LIN {X 0,Y 406.428,Z 396.116,A -85,B 0,C 180,E1 17978.8,E2 17978.8} C_VEL
LIN {X 0,Y 408.276,Z 399.712,A -85,B 0,C 180,E1 17977.389,E2 17977.389} C_VEL
LIN {X 0,Y 411.856,Z 402.645,A -85,B 0,C 180,E1 17975.473,E2 17975.473} C_VEL
LIN {X 0,Y 414.278,Z 406.426,A -85,B 0,C 180,E1 17974.252,E2 17974.252} C_VEL
LIN {X 0,Y 416.644,Z 408.719,A -85,B 0,C 180,E1 17973.259,E2 17973.259} C_VEL
LIN {X 0,Y 420.794,Z 414.411,A -85,B 0,C 180,E1 17971.588,E2 17971.588} C_VEL
LIN {X 0,Y 424.606,Z 419.568,A -85,B 0,C 180,E1 17970.247,E2 17970.247} C_VEL
LIN {X 0,Y 430.468,Z 427.804,A -85,B 0,C 180,E1 17968.376,E2 17968.376} C_VEL
LIN {X 0,Y 437.911,Z 439.101,A -85,B 0,C 180,E1 17966.262,E2 17966.262} C_VEL
LIN {X 0,Y 445.629,Z 451.395,A -85,B 0,C 180,E1 17964.313,E2 17964.313} C_VEL
LIN {X 0,Y 451.863,Z 462.203,A -85,B 0,C 180,E1 17962.861,E2 17962.861} C_VEL
LIN {X 0,Y 443.06,Z 655.512,A -85,B 0,C 180,E1 17959.181,E2 17959.181} C_VEL
LIN {X 0,Y 439.484,Z 737.589,A -85,B 0,C 180,E1 17957.617,E2 17957.617} C_VEL
LIN {X 0,Y 437.318,Z 760.996,A -85,B 0,C 180,E1 17956.985,E2 17956.985} C_VEL
LIN {X 0,Y 434.644,Z 783.7,A -85,B 0,C 180,E1 17956.155,E2 17956.155} C_VEL
LIN {X 0,Y 431.569,Z 804.772,A -85,B 0,C 180,E1 17955.152,E2 17955.152} C_VEL
LIN {X 0,Y 427.742,Z 827.839,A -85,B 0,C 180,E1 17953.785,E2 17953.785} C_VEL
LIN {X 0,Y 424.132,Z 847.133,A -85,B 0,C 180,E1 17952.397,E2 17952.397} C_VEL
LIN {X 0,Y 419.735,Z 868.682,A -85,B 0,C 180,E1 17950.546,E2 17950.546} C_VEL
LIN {X 0,Y 415.658,Z 887.581,A -85,B 0,C 180,E1 17948.629,E2 17948.629} C_VEL
LIN {X 0,Y 411.63,Z 905.465,A -85,B 0,C 180,E1 17946.487,E2 17946.487} C_VEL
LIN {X 0,Y 407.694,Z 922.843,A -85,B 0,C 180,E1 17944.086,E2 17944.086} C_VEL
LIN {X 0,Y 404.06,Z 938.881,A -85,B 0,C 180,E1 17941.479,E2 17941.479} C_VEL
LIN {X 0,Y 400.612,Z 954.751,A -85,B 0,C 180,E1 17938.474,E2 17938.474} C_VEL
LIN {X 0,Y 398,Z 967.71,A -85,B 0,C 180,E1 17935.605,E2 17935.605} C_VEL
LIN {X 0,Y 395.868,Z 979.3,A -85,B 0,C 180,E1 17932.58,E2 17932.58} C_VEL
LIN {X 0,Y 394.308,Z 989.212,A -85,B 0,C 180,E1 17929.559,E2 17929.559} C_VEL
LIN {X 0,Y 393.186,Z 997.751,A -85,B 0,C 180,E1 17926.4,E2 17926.4} C_VEL
LIN {X 0,Y 392.495,Z 1004.747,A -85,B 0,C 180,E1 17923.258,E2 17923.258} C_VEL
LIN {X 0,Y 392.089,Z 1010.305,A -85,B 0,C 180,E1 17919.99,E2 17919.99} C_VEL
LIN {X 0,Y 391.942,Z 1013.857,A -85,B 0,C 180,E1 17917.185,E2 17917.185} C_VEL
LIN {X 0,Y 391.914,Z 1016.519,A -85,B 0,C 180,E1 17913.954,E2 17913.954} C_VEL
LIN {X 0,Y 391.905,Z 1017.533,A -85,B 0,C 180,E1 17911.174,E2 17911.174} C_VEL
LIN {X 0,Y 391.911,Z 1017.466,A -85,B 0,C 180,E1 17908.396,E2 17908.396} C_VEL
LIN {X 0,Y 391.918,Z 1015.846,A -85,B 0,C 180,E1 17905.029,E2 17905.029} C_VEL
LIN {X 0,Y 391.977,Z 1013.229,A -85,B 0,C 180,E1 17902.235,E2 17902.235} C_VEL
LIN {X 0,Y 392.181,Z 1009.071,A -85,B 0,C 180,E1 17899.13,E2 17899.13} C_VEL
LIN {X 0,Y 392.616,Z 1003.242,A -85,B 0,C 180,E1 17895.993,E2 17895.993} C_VEL
LIN {X 0,Y 393.401,Z 996.051,A -85,B 0,C 180,E1 17892.858,E2 17892.858} C_VEL
LIN {X 0,Y 394.64,Z 987.03,A -85,B 0,C 180,E1 17889.695,E2 17889.695} C_VEL
LIN {X 0,Y 396.359,Z 976.876,A -85,B 0,C 180,E1 17886.667,E2 17886.667} C_VEL
LIN {X 0,Y 398.648,Z 964.781,A -85,B 0,C 180,E1 17883.651,E2 17883.651} C_VEL
LIN {X 0,Y 401.452,Z 951.514,A -85,B 0,C 180,E1 17880.787,E2 17880.787} C_VEL
LIN {X 0,Y 404.687,Z 936.825,A -85,B 0,C 180,E1 17878.087,E2 17878.087} C_VEL
LIN {X 0,Y 408.687,Z 919.41,A -85,B 0,C 180,E1 17875.339,E2 17875.339} C_VEL
LIN {X 0,Y 412.435,Z 903.112,A -85,B 0,C 180,E1 17873.13,E2 17873.13} C_VEL
LIN {X 0,Y 416.65,Z 884.299,A -85,B 0,C 180,E1 17870.951,E2 17870.951} C_VEL
LIN {X 0,Y 420.873,Z 864.938,A -85,B 0,C 180,E1 17869.036,E2 17869.036} C_VEL
LIN {X 0,Y 424.917,Z 844.471,A -85,B 0,C 180,E1 17867.345,E2 17867.345} C_VEL
LIN {X 0,Y 428.827,Z 823.074,A -85,B 0,C 180,E1 17865.862,E2 17865.862} C_VEL
LIN {X 0,Y 432.119,Z 802.52,A -85,B 0,C 180,E1 17864.7,E2 17864.7} C_VEL
LIN {X 0,Y 435.408,Z 778.669,A -85,B 0,C 180,E1 17863.628,E2 17863.628} C_VEL
LIN {X 0,Y 437.702,Z 758.039,A -85,B 0,C 180,E1 17862.917,E2 17862.917} C_VEL
LIN {X 0,Y 439.633,Z 733.719,A -85,B 0,C 180,E1 17862.311,E2 17862.311} C_VEL
LIN {X 0,Y 448.195,Z 525.035,A -85,B 0,C 180,E1 17858.416,E2 17858.416} C_VEL
LIN {X 0,Y 450.801,Z 461.932,A -85,B 0,C 180,E1 17857.207,E2 17857.207} C_VEL
LIN {X 0,Y 440.409,Z 445.676,A -85,B 0,C 180,E1 17855.016,E2 17855.016} C_VEL
LIN {X 0,Y 429.506,Z 429.721,A -85,B 0,C 180,E1 17852.53,E2 17852.53} C_VEL
LIN {X 0,Y 418.728,Z 414.832,A -85,B 0,C 180,E1 17849.819,E2 17849.819} C_VEL
LIN {X 0,Y 410.778,Z 404.455,A -85,B 0,C 180,E1 17847.625,E2 17847.625} C_VEL
LIN {X 0,Y 406.148,Z 398.624,A -85,B 0,C 180,E1 17846.263,E2 17846.263} C_VEL
LIN {X 0,Y 402.102,Z 393.64,A -85,B 0,C 180,E1 17845.006,E2 17845.006} C_VEL
LIN {X 0,Y 398.857,Z 389.644,A -85,B 0,C 180,E1 17843.96,E2 17843.96} C_VEL
LIN {X 0,Y 397.676,Z 388.128,A -85,B 0,C 180,E1 17843.563,E2 17843.563} C_VEL
LIN {X 0,Y 394.873,Z 385.623,A -85,B 0,C 180,E1 17842.636,E2 17842.636} C_VEL
LIN {X 0,Y 393.655,Z 382.808,A -85,B 0,C 180,E1 17842.034,E2 17842.034} C_VEL
LIN {X 0,Y 393.526,Z 382.083,A -85,B 0,C 180,E1 17841.461,E2 17841.461} C_VEL
LIN {X 0,Y 393.528,Z 382.017,A -85,B 0,C 180,E1 17837.446,E2 17837.446} C_VEL
LIN {X 0,Y 393.545,Z 382.024,A -85,B 0,C 180,E1 17833.517,E2 17833.517} C_VEL
LIN {X 0,Y 393.537,Z 382.019,A -85,B 0,C 180,E1 17829.505,E2 17829.505} C_VEL
LIN {X 0,Y 393.517,Z 382.017,A -85,B 0,C 180,E1 17825.686,E2 17825.686} C_VEL
LIN {X 0,Y 393.511,Z 382.017,A -85,B 0,C 180,E1 17821.747,E2 17821.747} C_VEL
LIN {X 0,Y 393.504,Z 382.024,A -85,B 0,C 180,E1 17817.961,E2 17817.961} C_VEL
LIN {X 0,Y 393.507,Z 382.031,A -85,B 0,C 180,E1 17814.02,E2 17814.02} C_VEL
LIN {X 0,Y 393.514,Z 382.03,A -85,B 0,C 180,E1 17810.05,E2 17810.05} C_VEL
LIN {X 0,Y 393.528,Z 382.024,A -85,B 0,C 180,E1 17806.182,E2 17806.182} C_VEL
LIN {X 0,Y 393.545,Z 382.014,A -85,B 0,C 180,E1 17802.294,E2 17802.294} C_VEL
LIN {X 0,Y 393.567,Z 382.01,A -85,B 0,C 180,E1 17798.384,E2 17798.384} C_VEL
LIN {X 0,Y 393.56,Z 382.013,A -85,B 0,C 180,E1 17794.393,E2 17794.393} C_VEL
LIN {X 0,Y 393.558,Z 382.018,A -85,B 0,C 180,E1 17790.47,E2 17790.47} C_VEL
LIN {X 0,Y 393.546,Z 382.028,A -85,B 0,C 180,E1 17786.542,E2 17786.542} C_VEL
LIN {X 0,Y 393.537,Z 382.019,A -85,B 0,C 180,E1 17782.61,E2 17782.61} C_VEL
LIN {X 0,Y 393.532,Z 382.015,A -85,B 0,C 180,E1 17778.759,E2 17778.759} C_VEL
LIN {X 0,Y 393.533,Z 382.024,A -85,B 0,C 180,E1 17774.723,E2 17774.723} C_VEL
LIN {X 0,Y 393.534,Z 382.018,A -85,B 0,C 180,E1 17770.758,E2 17770.758} C_VEL
LIN {X 0,Y 393.613,Z 382.321,A -85,B 0,C 180,E1 17769.416,E2 17769.416} C_VEL
LIN {X 0,Y 393.952,Z 383.729,A -85,B 0,C 180,E1 17769.046,E2 17769.046} C_VEL
LIN {X 0,Y 395.637,Z 386.503,A -85,B 0,C 180,E1 17768.423,E2 17768.423} C_VEL
LIN {X 0,Y 398.831,Z 388.927,A -85,B 0,C 180,E1 17767.401,E2 17767.401} C_VEL
LIN {X 0,Y 401.009,Z 392.541,A -85,B 0,C 180,E1 17766.655,E2 17766.655} C_VEL
LIN {X 0,Y 404.151,Z 395.276,A -85,B 0,C 180,E1 17765.715,E2 17765.715} C_VEL
LIN {X 0,Y 406.926,Z 399.204,A -85,B 0,C 180,E1 17764.847,E2 17764.847} C_VEL
LIN {X 0,Y 409.166,Z 401.398,A -85,B 0,C 180,E1 17764.205,E2 17764.205} C_VEL
LIN {X 0,Y 412.49,Z 405.713,A -85,B 0,C 180,E1 17763.251,E2 17763.251} C_VEL
LIN {X 0,Y 414.192,Z 407.663,A -85,B 0,C 180,E1 17762.788,E2 17762.788} C_VEL
LIN {X 0,Y 419.544,Z 414.327,A -85,B 0,C 180,E1 17761.373,E2 17761.373} C_VEL
LIN {X 0,Y 423.817,Z 419.73,A -85,B 0,C 180,E1 17760.292,E2 17760.292} C_VEL
LIN {X 0,Y 432.407,Z 430.894,A -85,B 0,C 180,E1 17758.237,E2 17758.237} C_VEL
LIN {X 0,Y 443.538,Z 446.105,A -85,B 0,C 180,E1 17755.797,E2 17755.797} C_VEL
LIN {X 0,Y 450.635,Z 456.669,A -85,B 0,C 180,E1 17754.337,E2 17754.337} C_VEL
LIN {X 0,Y 441.914,Z 664.576,A -85,B 0,C 180,E1 17750.46,E2 17750.46} C_VEL
LIN {X 0,Y 441.065,Z 686.182,A -85,B 0,C 180,E1 17750.061,E2 17750.061} C_VEL
LIN {X 0,Y 440.083,Z 693.883,A -85,B 0,C 180,E1 17750.016,E2 17750.016} C_VEL
LIN {X 0,Y 434.779,Z 714.411,A -85,B 0,C 180,E1 17750.219,E2 17750.219} C_VEL
LIN {X 0,Y 433.809,Z 720.955,A -85,B 0,C 180,E1 17750.126,E2 17750.126} C_VEL
LIN {X 0,Y 431.867,Z 741.999,A -85,B 0,C 180,E1 17749.509,E2 17749.509} C_VEL
LIN {X 0,Y 429.108,Z 764.775,A -85,B 0,C 180,E1 17748.611,E2 17748.611} C_VEL
LIN {X 0,Y 426.34,Z 783.59,A -85,B 0,C 180,E1 17747.675,E2 17747.675} C_VEL
LIN {X 0,Y 422.604,Z 805.364,A -85,B 0,C 180,E1 17746.348,E2 17746.348} C_VEL
LIN {X 0,Y 419.031,Z 823.676,A -85,B 0,C 180,E1 17745,E2 17745} C_VEL
LIN {X 0,Y 414.557,Z 844.411,A -85,B 0,C 180,E1 17743.183,E2 17743.183} C_VEL
LIN {X 0,Y 410.383,Z 862.505,A -85,B 0,C 180,E1 17741.306,E2 17741.306} C_VEL
LIN {X 0,Y 406.042,Z 880.264,A -85,B 0,C 180,E1 17739.134,E2 17739.134} C_VEL
LIN {X 0,Y 402.007,Z 896.346,A -85,B 0,C 180,E1 17736.852,E2 17736.852} C_VEL
LIN {X 0,Y 398.055,Z 911.792,A -85,B 0,C 180,E1 17734.275,E2 17734.275} C_VEL
LIN {X 0,Y 394.61,Z 925.735,A -85,B 0,C 180,E1 17731.593,E2 17731.593} C_VEL
LIN {X 0,Y 391.538,Z 938.518,A -85,B 0,C 180,E1 17728.679,E2 17728.679} C_VEL
LIN {X 0,Y 388.972,Z 950.224,A -85,B 0,C 180,E1 17725.573,E2 17725.573} C_VEL
LIN {X 0,Y 387.022,Z 960.112,A -85,B 0,C 180,E1 17722.425,E2 17722.425} C_VEL
LIN {X 0,Y 385.538,Z 969.205,A -85,B 0,C 180,E1 17718.931,E2 17718.931} C_VEL
LIN {X 0,Y 384.68,Z 975.978,A -85,B 0,C 180,E1 17715.7,E2 17715.7} C_VEL
LIN {X 0,Y 384.188,Z 981.504,A -85,B 0,C 180,E1 17712.268,E2 17712.268} C_VEL
LIN {X 0,Y 383.982,Z 985.352,A -85,B 0,C 180,E1 17708.936,E2 17708.936} C_VEL
LIN {X 0,Y 383.929,Z 987.716,A -85,B 0,C 180,E1 17705.535,E2 17705.535} C_VEL
LIN {X 0,Y 383.908,Z 988.577,A -85,B 0,C 180,E1 17702.315,E2 17702.315} C_VEL
LIN {X 0,Y 383.929,Z 987.981,A -85,B 0,C 180,E1 17698.955,E2 17698.955} C_VEL
LIN {X 0,Y 383.955,Z 985.95,A -85,B 0,C 180,E1 17695.588,E2 17695.588} C_VEL
LIN {X 0,Y 384.133,Z 982.409,A -85,B 0,C 180,E1 17692.285,E2 17692.285} C_VEL
LIN {X 0,Y 384.541,Z 977.393,A -85,B 0,C 180,E1 17688.942,E2 17688.942} C_VEL
LIN {X 0,Y 385.364,Z 970.543,A -85,B 0,C 180,E1 17685.522,E2 17685.522} C_VEL
LIN {X 0,Y 386.671,Z 962.482,A -85,B 0,C 180,E1 17682.247,E2 17682.247} C_VEL
LIN {X 0,Y 388.536,Z 952.579,A -85,B 0,C 180,E1 17678.994,E2 17678.994} C_VEL
LIN {X 0,Y 391.128,Z 940.768,A -85,B 0,C 180,E1 17675.723,E2 17675.723} C_VEL
LIN {X 0,Y 394.033,Z 928.538,A -85,B 0,C 180,E1 17672.865,E2 17672.865} C_VEL
LIN {X 0,Y 397.816,Z 913.455,A -85,B 0,C 180,E1 17669.87,E2 17669.87} C_VEL
LIN {X 0,Y 401.794,Z 898.064,A -85,B 0,C 180,E1 17667.251,E2 17667.251} C_VEL
LIN {X 0,Y 405.906,Z 881.802,A -85,B 0,C 180,E1 17664.912,E2 17664.912} C_VEL
LIN {X 0,Y 410.309,Z 864.198,A -85,B 0,C 180,E1 17662.721,E2 17662.721} C_VEL
LIN {X 0,Y 414.446,Z 846.464,A -85,B 0,C 180,E1 17660.853,E2 17660.853} C_VEL
LIN {X 0,Y 418.988,Z 825.858,A -85,B 0,C 180,E1 17659.011,E2 17659.011} C_VEL
LIN {X 0,Y 422.741,Z 806.937,A -85,B 0,C 180,E1 17657.598,E2 17657.598} C_VEL
LIN {X 0,Y 426.635,Z 784.75,A -85,B 0,C 180,E1 17656.229,E2 17656.229} C_VEL
LIN {X 0,Y 429.41,Z 766.27,A -85,B 0,C 180,E1 17655.298,E2 17655.298} C_VEL
LIN {X 0,Y 432.256,Z 743.229,A -85,B 0,C 180,E1 17654.377,E2 17654.377} C_VEL
LIN {X 0,Y 434.174,Z 722.916,A -85,B 0,C 180,E1 17653.771,E2 17653.771} C_VEL
LIN {X 0,Y 435.95,Z 691.902,A -85,B 0,C 180,E1 17653.119,E2 17653.119} C_VEL
LIN {X 0,Y 445.434,Z 492.104,A -85,B 0,C 180,E1 17649.297,E2 17649.297} C_VEL
LIN {X 0,Y 446.947,Z 460.775,A -85,B 0,C 180,E1 17648.669,E2 17648.669} C_VEL
LIN {X 0,Y 438.774,Z 448.403,A -85,B 0,C 180,E1 17646.674,E2 17646.674} C_VEL
LIN {X 0,Y 430.575,Z 436.674,A -85,B 0,C 180,E1 17644.429,E2 17644.429} C_VEL
LIN {X 0,Y 425.629,Z 430.22,A -85,B 0,C 180,E1 17642.916,E2 17642.916} C_VEL
LIN {X 0,Y 422.462,Z 426.015,A -85,B 0,C 180,E1 17641.865,E2 17641.865} C_VEL
LIN {X 0,Y 418.675,Z 421.042,A -85,B 0,C 180,E1 17640.479,E2 17640.479} C_VEL
LIN {X 0,Y 415.228,Z 416.743,A -85,B 0,C 180,E1 17639.104,E2 17639.104} C_VEL
LIN {X 0,Y 414.077,Z 415.376,A -85,B 0,C 180,E1 17638.608,E2 17638.608} C_VEL
LIN {X 0,Y 410.92,Z 411.698,A -85,B 0,C 180,E1 17637.107,E2 17637.107} C_VEL
LIN {X 0,Y 409.736,Z 409.74,A -85,B 0,C 180,E1 17636.465,E2 17636.465} C_VEL
LIN {X 0,Y 406.459,Z 406.882,A -85,B 0,C 180,E1 17634.566,E2 17634.566} C_VEL
LIN {X 0,Y 404.667,Z 403.582,A -85,B 0,C 180,E1 17633.189,E2 17633.189} C_VEL
LIN {X 0,Y 400.609,Z 400.405,A -85,B 0,C 180,E1 17628.483,E2 17628.483} C_VEL
LIN {X 0,Y 400.207,Z 399.651,A -85,B 0,C 180,E1 17625.976,E2 17625.976} C_VEL
LIN {X 0,Y 400.964,Z 400.936,A -85,B 0,C 180,E1 17623.187,E2 17623.187} C_VEL
LIN {X 0,Y 405.042,Z 404.041,A -85,B 0,C 180,E1 17618.985,E2 17618.985} C_VEL
LIN {X 0,Y 406.914,Z 407.563,A -85,B 0,C 180,E1 17617.53,E2 17617.53} C_VEL
LIN {X 0,Y 410.102,Z 410.218,A -85,B 0,C 180,E1 17615.783,E2 17615.783} C_VEL
LIN {X 0,Y 412.806,Z 414.296,A -85,B 0,C 180,E1 17614.384,E2 17614.384} C_VEL
LIN {X 0,Y 414.826,Z 416.366,A -85,B 0,C 180,E1 17613.519,E2 17613.519} C_VEL
LIN {X 0,Y 418.809,Z 421.973,A -85,B 0,C 180,E1 17611.868,E2 17611.868} C_VEL
LIN {X 0,Y 422.265,Z 426.738,A -85,B 0,C 180,E1 17610.616,E2 17610.616} C_VEL
LIN {X 0,Y 427.794,Z 434.728,A -85,B 0,C 180,E1 17608.784,E2 17608.784} C_VEL
LIN {X 0,Y 435.211,Z 446.196,A -85,B 0,C 180,E1 17606.618,E2 17606.618} C_VEL
LIN {X 0,Y 443.39,Z 459.583,A -85,B 0,C 180,E1 17604.499,E2 17604.499} C_VEL
LIN {X 0,Y 447.005,Z 466.235,A -85,B 0,C 180,E1 17603.619,E2 17603.619} C_VEL
LIN {X 0,Y 437.783,Z 657.986,A -85,B 0,C 180,E1 17599.933,E2 17599.933} C_VEL
LIN {X 0,Y 434.097,Z 737.688,A -85,B 0,C 180,E1 17598.396,E2 17598.396} C_VEL
LIN {X 0,Y 431.819,Z 761.162,A -85,B 0,C 180,E1 17597.754,E2 17597.754} C_VEL
LIN {X 0,Y 428.968,Z 784.037,A -85,B 0,C 180,E1 17596.907,E2 17596.907} C_VEL
LIN {X 0,Y 425.651,Z 805.681,A -85,B 0,C 180,E1 17595.862,E2 17595.862} C_VEL
LIN {X 0,Y 421.685,Z 828.309,A -85,B 0,C 180,E1 17594.499,E2 17594.499} C_VEL
LIN {X 0,Y 417.893,Z 847.639,A -85,B 0,C 180,E1 17593.089,E2 17593.089} C_VEL
LIN {X 0,Y 413.338,Z 868.814,A -85,B 0,C 180,E1 17591.24,E2 17591.24} C_VEL
LIN {X 0,Y 409.022,Z 887.843,A -85,B 0,C 180,E1 17589.285,E2 17589.285} C_VEL
LIN {X 0,Y 404.67,Z 906.087,A -85,B 0,C 180,E1 17587.055,E2 17587.055} C_VEL
LIN {X 0,Y 400.525,Z 923.381,A -85,B 0,C 180,E1 17584.609,E2 17584.609} C_VEL
LIN {X 0,Y 396.9,Z 938.465,A -85,B 0,C 180,E1 17582.114,E2 17582.114} C_VEL
LIN {X 0,Y 393.234,Z 954.35,A -85,B 0,C 180,E1 17579.059,E2 17579.059} C_VEL
LIN {X 0,Y 390.582,Z 966.668,A -85,B 0,C 180,E1 17576.291,E2 17576.291} C_VEL
LIN {X 0,Y 388.169,Z 978.931,A -85,B 0,C 180,E1 17573.053,E2 17573.053} C_VEL
LIN {X 0,Y 386.49,Z 988.853,A -85,B 0,C 180,E1 17569.971,E2 17569.971} C_VEL
LIN {X 0,Y 385.283,Z 997.406,A -85,B 0,C 180,E1 17566.746,E2 17566.746} C_VEL
LIN {X 0,Y 384.564,Z 1004.101,A -85,B 0,C 180,E1 17563.69,E2 17563.69} C_VEL
LIN {X 0,Y 384.113,Z 1009.865,A -85,B 0,C 180,E1 17560.284,E2 17560.284} C_VEL
LIN {X 0,Y 383.956,Z 1013.377,A -85,B 0,C 180,E1 17557.486,E2 17557.486} C_VEL
LIN {X 0,Y 383.918,Z 1016.142,A -85,B 0,C 180,E1 17554.186,E2 17554.186} C_VEL
LIN {X 0,Y 383.911,Z 1017.231,A -85,B 0,C 180,E1 17551.198,E2 17551.198} C_VEL
LIN {X 0,Y 383.916,Z 1017.167,A -85,B 0,C 180,E1 17548.363,E2 17548.363} C_VEL
LIN {X 0,Y 383.923,Z 1015.548,A -85,B 0,C 180,E1 17544.925,E2 17544.925} C_VEL
LIN {X 0,Y 384.008,Z 1012.766,A -85,B 0,C 180,E1 17541.922,E2 17541.922} C_VEL
LIN {X 0,Y 384.239,Z 1007.992,A -85,B 0,C 180,E1 17538.447,E2 17538.447} C_VEL
LIN {X 0,Y 384.73,Z 1002.337,A -85,B 0,C 180,E1 17535.404,E2 17535.404} C_VEL
LIN {X 0,Y 385.685,Z 994.537,A -85,B 0,C 180,E1 17532.037,E2 17532.037} C_VEL
LIN {X 0,Y 387.024,Z 985.772,A -85,B 0,C 180,E1 17528.961,E2 17528.961} C_VEL
LIN {X 0,Y 389.148,Z 974.254,A -85,B 0,C 180,E1 17525.571,E2 17525.571} C_VEL
LIN {X 0,Y 391.585,Z 962.5,A -85,B 0,C 180,E1 17522.645,E2 17522.645} C_VEL
LIN {X 0,Y 394.843,Z 948.018,A -85,B 0,C 180,E1 17519.578,E2 17519.578} C_VEL
LIN {X 0,Y 398.536,Z 932.669,A -85,B 0,C 180,E1 17516.787,E2 17516.787} C_VEL
LIN {X 0,Y 402.43,Z 916.445,A -85,B 0,C 180,E1 17514.284,E2 17514.284} C_VEL
LIN {X 0,Y 406.754,Z 898.616,A -85,B 0,C 180,E1 17511.91,E2 17511.91} C_VEL
LIN {X 0,Y 410.829,Z 881.207,A -85,B 0,C 180,E1 17509.937,E2 17509.937} C_VEL
LIN {X 0,Y 415.463,Z 860.345,A -85,B 0,C 180,E1 17507.922,E2 17507.922} C_VEL
LIN {X 0,Y 419.428,Z 841.214,A -85,B 0,C 180,E1 17506.368,E2 17506.368} C_VEL
LIN {X 0,Y 423.486,Z 819.472,A -85,B 0,C 180,E1 17504.905,E2 17504.905} C_VEL
LIN {X 0,Y 427.068,Z 797.92,A -85,B 0,C 180,E1 17503.718,E2 17503.718} C_VEL
LIN {X 0,Y 430.038,Z 776.108,A -85,B 0,C 180,E1 17502.776,E2 17502.776} C_VEL
LIN {X 0,Y 432.538,Z 754.231,A -85,B 0,C 180,E1 17502.042,E2 17502.042} C_VEL
LIN {X 0,Y 434.294,Z 730.724,A -85,B 0,C 180,E1 17501.484,E2 17501.484} C_VEL
LIN {X 0,Y 443.269,Z 521.692,A -85,B 0,C 180,E1 17497.553,E2 17497.553} C_VEL
LIN {X 0,Y 445.703,Z 465.789,A -85,B 0,C 180,E1 17496.475,E2 17496.475} C_VEL
LIN {X 0,Y 435.041,Z 449.15,A -85,B 0,C 180,E1 17494.149,E2 17494.149} C_VEL
LIN {X 0,Y 425.183,Z 434.788,A -85,B 0,C 180,E1 17491.826,E2 17491.826} C_VEL
LIN {X 0,Y 415.533,Z 421.274,A -85,B 0,C 180,E1 17489.318,E2 17489.318} C_VEL
LIN {X 0,Y 407.875,Z 411.22,A -85,B 0,C 180,E1 17487.165,E2 17487.165} C_VEL
LIN {X 0,Y 403.321,Z 405.407,A -85,B 0,C 180,E1 17485.789,E2 17485.789} C_VEL
LIN {X 0,Y 399.612,Z 400.791,A -85,B 0,C 180,E1 17484.619,E2 17484.619} C_VEL
LIN {X 0,Y 395.945,Z 396.037,A -85,B 0,C 180,E1 17483.396,E2 17483.396} C_VEL
LIN {X 0,Y 392.41,Z 392.601,A -85,B 0,C 180,E1 17482.193,E2 17482.193} C_VEL
LIN {X 0,Y 390.723,Z 389.598,A -85,B 0,C 180,E1 17481.543,E2 17481.543} C_VEL
LIN {X 0,Y 387.439,Z 387.253,A -85,B 0,C 180,E1 17480.388,E2 17480.388} C_VEL
LIN {X 0,Y 385.72,Z 383.756,A -85,B 0,C 180,E1 17479.535,E2 17479.535} C_VEL
LIN {X 0,Y 385.558,Z 383.051,A -85,B 0,C 180,E1 17478.914,E2 17478.914} C_VEL
LIN {X 0,Y 385.565,Z 383.008,A -85,B 0,C 180,E1 17475.029,E2 17475.029} C_VEL
LIN {X 0,Y 385.588,Z 383.006,A -85,B 0,C 180,E1 17471.214,E2 17471.214} C_VEL
LIN {X 0,Y 385.602,Z 383.015,A -85,B 0,C 180,E1 17467.149,E2 17467.149} C_VEL
LIN {X 0,Y 385.602,Z 383.008,A -85,B 0,C 180,E1 17463.121,E2 17463.121} C_VEL
LIN {X 0,Y 385.614,Z 383.001,A -85,B 0,C 180,E1 17459.108,E2 17459.108} C_VEL
LIN {X 0,Y 385.606,Z 383.003,A -85,B 0,C 180,E1 17455.091,E2 17455.091} C_VEL
LIN {X 0,Y 385.595,Z 383.006,A -85,B 0,C 180,E1 17451.199,E2 17451.199} C_VEL
LIN {X 0,Y 385.586,Z 383.015,A -85,B 0,C 180,E1 17447.266,E2 17447.266} C_VEL
LIN {X 0,Y 385.578,Z 383.02,A -85,B 0,C 180,E1 17443.426,E2 17443.426} C_VEL
LIN {X 0,Y 385.58,Z 383.014,A -85,B 0,C 180,E1 17439.391,E2 17439.391} C_VEL
LIN {X 0,Y 385.579,Z 383.006,A -85,B 0,C 180,E1 17435.323,E2 17435.323} C_VEL
LIN {X 0,Y 385.583,Z 383.003,A -85,B 0,C 180,E1 17431.332,E2 17431.332} C_VEL
LIN {X 0,Y 385.589,Z 383.01,A -85,B 0,C 180,E1 17427.359,E2 17427.359} C_VEL
LIN {X 0,Y 385.597,Z 383.018,A -85,B 0,C 180,E1 17423.387,E2 17423.387} C_VEL
LIN {X 0,Y 385.605,Z 383.004,A -85,B 0,C 180,E1 17419.395,E2 17419.395} C_VEL
LIN {X 0,Y 385.61,Z 383.003,A -85,B 0,C 180,E1 17415.357,E2 17415.357} C_VEL
LIN {X 0,Y 385.661,Z 383.299,A -85,B 0,C 180,E1 17411.973,E2 17411.973} C_VEL
LIN {X 0,Y 386.02,Z 384.671,A -85,B 0,C 180,E1 17411.527,E2 17411.527} C_VEL
LIN {X 0,Y 387.738,Z 387.532,A -85,B 0,C 180,E1 17410.812,E2 17410.812} C_VEL
LIN {X 0,Y 391.046,Z 389.934,A -85,B 0,C 180,E1 17409.65,E2 17409.65} C_VEL
LIN {X 0,Y 393.067,Z 393.427,A -85,B 0,C 180,E1 17408.886,E2 17408.886} C_VEL
LIN {X 0,Y 396.358,Z 396.252,A -85,B 0,C 180,E1 17407.799,E2 17407.799} C_VEL
LIN {X 0,Y 399.057,Z 400.215,A -85,B 0,C 180,E1 17406.879,E2 17406.879} C_VEL
LIN {X 0,Y 401.715,Z 402.679,A -85,B 0,C 180,E1 17406.069,E2 17406.069} C_VEL
LIN {X 0,Y 404.956,Z 406.856,A -85,B 0,C 180,E1 17405.065,E2 17405.065} C_VEL
LIN {X 0,Y 406.693,Z 408.75,A -85,B 0,C 180,E1 17404.552,E2 17404.552} C_VEL
LIN {X 0,Y 410.478,Z 413.367,A -85,B 0,C 180,E1 17403.459,E2 17403.459} C_VEL
LIN {X 0,Y 420.192,Z 425.608,A -85,B 0,C 180,E1 17400.866,E2 17400.866} C_VEL
LIN {X 0,Y 431.442,Z 440.478,A -85,B 0,C 180,E1 17398.138,E2 17398.138} C_VEL
LIN {X 0,Y 443.192,Z 457.042,A -85,B 0,C 180,E1 17395.559,E2 17395.559} C_VEL
LIN {X 0,Y 445.503,Z 460.776,A -85,B 0,C 180,E1 17395.069,E2 17395.069} C_VEL
LIN {X 0,Y 436.352,Z 669.306,A -85,B 0,C 180,E1 17391.15,E2 17391.15} C_VEL
LIN {X 0,Y 434.124,Z 717.19,A -85,B 0,C 180,E1 17390.223,E2 17390.223} C_VEL
LIN {X 0,Y 433.809,Z 720.955,A -85,B 0,C 180,E1 17390.126,E2 17390.126} C_VEL
LIN {X 0,Y 432.442,Z 728.564,A -85,B 0,C 180,E1 17390.036,E2 17390.036} C_VEL
LIN {X 0,Y 426.299,Z 747.731,A -85,B 0,C 180,E1 17390.024,E2 17390.024} C_VEL
LIN {X 0,Y 424.81,Z 755.185,A -85,B 0,C 180,E1 17389.809,E2 17389.809} C_VEL
LIN {X 0,Y 421.501,Z 778.336,A -85,B 0,C 180,E1 17388.744,E2 17388.744} C_VEL
LIN {X 0,Y 417.955,Z 799.173,A -85,B 0,C 180,E1 17387.538,E2 17387.538} C_VEL
LIN {X 0,Y 413.828,Z 820.109,A -85,B 0,C 180,E1 17386.055,E2 17386.055} C_VEL
LIN {X 0,Y 409.772,Z 838.808,A -85,B 0,C 180,E1 17384.479,E2 17384.479} C_VEL
LIN {X 0,Y 405.135,Z 858.13,A -85,B 0,C 180,E1 17382.539,E2 17382.539} C_VEL
LIN {X 0,Y 400.618,Z 876.151,A -85,B 0,C 180,E1 17380.42,E2 17380.42} C_VEL
LIN {X 0,Y 396.248,Z 892.644,A -85,B 0,C 180,E1 17378.119,E2 17378.119} C_VEL
LIN {X 0,Y 392.03,Z 908.525,A -85,B 0,C 180,E1 17375.557,E2 17375.557} C_VEL
LIN {X 0,Y 388.165,Z 922.99,A -85,B 0,C 180,E1 17372.801,E2 17372.801} C_VEL
LIN {X 0,Y 384.455,Z 937.496,A -85,B 0,C 180,E1 17369.548,E2 17369.548} C_VEL
LIN {X 0,Y 381.649,Z 949.412,A -85,B 0,C 180,E1 17366.391,E2 17366.391} C_VEL
LIN {X 0,Y 379.497,Z 959.438,A -85,B 0,C 180,E1 17363.187,E2 17363.187} C_VEL
LIN {X 0,Y 377.901,Z 968.388,A -85,B 0,C 180,E1 17359.785,E2 17359.785} C_VEL
LIN {X 0,Y 376.887,Z 975.289,A -85,B 0,C 180,E1 17356.495,E2 17356.495} C_VEL
LIN {X 0,Y 376.282,Z 981.105,A -85,B 0,C 180,E1 17353.001,E2 17353.001} C_VEL
LIN {X 0,Y 376.034,Z 984.954,A -85,B 0,C 180,E1 17349.774,E2 17349.774} C_VEL
LIN {X 0,Y 375.921,Z 987.6,A -85,B 0,C 180,E1 17346.483,E2 17346.483} C_VEL
LIN {X 0,Y 375.915,Z 988.737,A -85,B 0,C 180,E1 17343.284,E2 17343.284} C_VEL
LIN {X 0,Y 375.909,Z 988.705,A -85,B 0,C 180,E1 17340.344,E2 17340.344} C_VEL
LIN {X 0,Y 375.941,Z 987.282,A -85,B 0,C 180,E1 17336.907,E2 17336.907} C_VEL
LIN {X 0,Y 376.039,Z 984.684,A -85,B 0,C 180,E1 17333.819,E2 17333.819} C_VEL
LIN {X 0,Y 376.355,Z 980.422,A -85,B 0,C 180,E1 17330.382,E2 17330.382} C_VEL
LIN {X 0,Y 376.989,Z 974.724,A -85,B 0,C 180,E1 17327.056,E2 17327.056} C_VEL
LIN {X 0,Y 378.188,Z 966.823,A -85,B 0,C 180,E1 17323.425,E2 17323.425} C_VEL
LIN {X 0,Y 379.817,Z 958.221,A -85,B 0,C 180,E1 17320.229,E2 17320.229} C_VEL
LIN {X 0,Y 382.266,Z 947.064,A -85,B 0,C 180,E1 17316.797,E2 17316.797} C_VEL
LIN {X 0,Y 385.16,Z 935.351,A -85,B 0,C 180,E1 17313.748,E2 17313.748} C_VEL
LIN {X 0,Y 388.679,Z 921.716,A -85,B 0,C 180,E1 17310.768,E2 17310.768} C_VEL
LIN {X 0,Y 392.807,Z 906.532,A -85,B 0,C 180,E1 17307.928,E2 17307.928} C_VEL
LIN {X 0,Y 396.875,Z 891.423,A -85,B 0,C 180,E1 17305.519,E2 17305.519} C_VEL
LIN {X 0,Y 401.802,Z 872.874,A -85,B 0,C 180,E1 17302.998,E2 17302.998} C_VEL
LIN {X 0,Y 406.27,Z 855.442,A -85,B 0,C 180,E1 17300.983,E2 17300.983} C_VEL
LIN {X 0,Y 410.824,Z 836.233,A -85,B 0,C 180,E1 17299.108,E2 17299.108} C_VEL
LIN {X 0,Y 415.255,Z 816.101,A -85,B 0,C 180,E1 17297.445,E2 17297.445} C_VEL
LIN {X 0,Y 419.263,Z 795.229,A -85,B 0,C 180,E1 17296.032,E2 17296.032} C_VEL
LIN {X 0,Y 423.062,Z 772.693,A -85,B 0,C 180,E1 17294.789,E2 17294.789} C_VEL
LIN {X 0,Y 425.887,Z 752.197,A -85,B 0,C 180,E1 17293.895,E2 17293.895} C_VEL
LIN {X 0,Y 428.471,Z 728.496,A -85,B 0,C 180,E1 17293.109,E2 17293.109} C_VEL
LIN {X 0,Y 430.076,Z 706.892,A -85,B 0,C 180,E1 17292.596,E2 17292.596} C_VEL
LIN {X 0,Y 440.369,Z 500.943,A -85,B 0,C 180,E1 17288.617,E2 17288.617} C_VEL
LIN {X 0,Y 442.238,Z 464.937,A -85,B 0,C 180,E1 17287.894,E2 17287.894} C_VEL
LIN {X 0,Y 433.689,Z 451.973,A -85,B 0,C 180,E1 17285.69,E2 17285.69} C_VEL
LIN {X 0,Y 426.589,Z 441.93,A -85,B 0,C 180,E1 17283.629,E2 17283.629} C_VEL
LIN {X 0,Y 420.568,Z 433.629,A -85,B 0,C 180,E1 17281.635,E2 17281.635} C_VEL
LIN {X 0,Y 416.392,Z 428.208,A -85,B 0,C 180,E1 17280.069,E2 17280.069} C_VEL
LIN {X 0,Y 412.927,Z 423.552,A -85,B 0,C 180,E1 17278.613,E2 17278.613} C_VEL
LIN {X 0,Y 409.243,Z 419.35,A -85,B 0,C 180,E1 17276.849,E2 17276.849} C_VEL
LIN {X 0,Y 408.086,Z 417.423,A -85,B 0,C 180,E1 17276.208,E2 17276.208} C_VEL
LIN {X 0,Y 404.779,Z 414.277,A -85,B 0,C 180,E1 17274.188,E2 17274.188} C_VEL
LIN {X 0,Y 403.152,Z 411.298,A -85,B 0,C 180,E1 17272.877,E2 17272.877} C_VEL
LIN {X 0,Y 399.371,Z 408.062,A -85,B 0,C 180,E1 17268.007,E2 17268.007} C_VEL
LIN {X 0,Y 399.136,Z 407.651,A -85,B 0,C 180,E1 17265.641,E2 17265.641} C_VEL
LIN {X 0,Y 400.343,Z 409.394,A -85,B 0,C 180,E1 17262.411,E2 17262.411} C_VEL
LIN {X 0,Y 403.575,Z 411.758,A -85,B 0,C 180,E1 17259.251,E2 17259.251} C_VEL
LIN {X 0,Y 405.54,Z 415.384,A -85,B 0,C 180,E1 17257.686,E2 17257.686} C_VEL
LIN {X 0,Y 408.419,Z 417.888,A -85,B 0,C 180,E1 17256.061,E2 17256.061} C_VEL
LIN {X 0,Y 411.201,Z 422.009,A -85,B 0,C 180,E1 17254.586,E2 17254.586} C_VEL
LIN {X 0,Y 413.018,Z 423.995,A -85,B 0,C 180,E1 17253.781,E2 17253.781} C_VEL
LIN {X 0,Y 416.761,Z 429.392,A -85,B 0,C 180,E1 17252.185,E2 17252.185} C_VEL
LIN {X 0,Y 420.139,Z 434.206,A -85,B 0,C 180,E1 17250.917,E2 17250.917} C_VEL
LIN {X 0,Y 425.268,Z 441.814,A -85,B 0,C 180,E1 17249.167,E2 17249.167} C_VEL
LIN {X 0,Y 432.638,Z 453.448,A -85,B 0,C 180,E1 17246.948,E2 17246.948} C_VEL
LIN {X 0,Y 441.399,Z 468.266,A -85,B 0,C 180,E1 17244.623,E2 17244.623} C_VEL
LIN {X 0,Y 442.267,Z 470.23,A -85,B 0,C 180,E1 17244.396,E2 17244.396} C_VEL
LIN {X 0,Y 432.512,Z 662.131,A -85,B 0,C 180,E1 17240.672,E2 17240.672} C_VEL
LIN {X 0,Y 428.854,Z 737.152,A -85,B 0,C 180,E1 17239.21,E2 17239.21} C_VEL
LIN {X 0,Y 426.51,Z 760.474,A -85,B 0,C 180,E1 17238.571,E2 17238.571} C_VEL
LIN {X 0,Y 423.635,Z 782.793,A -85,B 0,C 180,E1 17237.749,E2 17237.749} C_VEL
LIN {X 0,Y 420.237,Z 804.101,A -85,B 0,C 180,E1 17236.727,E2 17236.727} C_VEL
LIN {X 0,Y 416.245,Z 826.089,A -85,B 0,C 180,E1 17235.419,E2 17235.419} C_VEL
LIN {X 0,Y 412.088,Z 846.347,A -85,B 0,C 180,E1 17233.946,E2 17233.946} C_VEL
LIN {X 0,Y 407.317,Z 867.682,A -85,B 0,C 180,E1 17232.082,E2 17232.082} C_VEL
LIN {X 0,Y 402.928,Z 886.074,A -85,B 0,C 180,E1 17230.183,E2 17230.183} C_VEL
LIN {X 0,Y 398.333,Z 904.393,A -85,B 0,C 180,E1 17227.954,E2 17227.954} C_VEL
LIN {X 0,Y 394.03,Z 921.537,A -85,B 0,C 180,E1 17225.531,E2 17225.531} C_VEL
LIN {X 0,Y 390.008,Z 937.199,A -85,B 0,C 180,E1 17222.926,E2 17222.926} C_VEL
LIN {X 0,Y 386.455,Z 951.796,A -85,B 0,C 180,E1 17220.131,E2 17220.131} C_VEL
LIN {X 0,Y 383.356,Z 964.975,A -85,B 0,C 180,E1 17217.161,E2 17217.161} C_VEL
LIN {X 0,Y 380.7,Z 977.499,A -85,B 0,C 180,E1 17213.861,E2 17213.861} C_VEL
LIN {X 0,Y 378.919,Z 987.073,A -85,B 0,C 180,E1 17210.873,E2 17210.873} C_VEL
LIN {X 0,Y 377.435,Z 996.698,A -85,B 0,C 180,E1 17207.264,E2 17207.264} C_VEL
LIN {X 0,Y 376.665,Z 1003.14,A -85,B 0,C 180,E1 17204.296,E2 17204.296} C_VEL
LIN {X 0,Y 376.163,Z 1009.234,A -85,B 0,C 180,E1 17200.727,E2 17200.727} C_VEL
LIN {X 0,Y 375.981,Z 1012.899,A -85,B 0,C 180,E1 17197.799,E2 17197.799} C_VEL
LIN {X 0,Y 375.918,Z 1015.681,A -85,B 0,C 180,E1 17194.581,E2 17194.581} C_VEL
LIN {X 0,Y 375.921,Z 1016.905,A -85,B 0,C 180,E1 17191.376,E2 17191.376} C_VEL
LIN {X 0,Y 375.922,Z 1016.892,A -85,B 0,C 180,E1 17188.481,E2 17188.481} C_VEL
LIN {X 0,Y 375.922,Z 1015.483,A -85,B 0,C 180,E1 17185.122,E2 17185.122} C_VEL
LIN {X 0,Y 375.996,Z 1012.795,A -85,B 0,C 180,E1 17182.057,E2 17182.057} C_VEL
LIN {X 0,Y 376.206,Z 1008.687,A -85,B 0,C 180,E1 17178.818,E2 17178.818} C_VEL
LIN {X 0,Y 376.697,Z 1002.964,A -85,B 0,C 180,E1 17175.557,E2 17175.557} C_VEL
LIN {X 0,Y 377.541,Z 996.155,A -85,B 0,C 180,E1 17172.433,E2 17172.433} C_VEL
LIN {X 0,Y 379.014,Z 986.863,A -85,B 0,C 180,E1 17168.981,E2 17168.981} C_VEL
LIN {X 0,Y 381.076,Z 976.252,A -85,B 0,C 180,E1 17165.68,E2 17165.68} C_VEL
LIN {X 0,Y 383.691,Z 964.107,A -85,B 0,C 180,E1 17162.539,E2 17162.539} C_VEL
LIN {X 0,Y 386.877,Z 950.806,A -85,B 0,C 180,E1 17159.572,E2 17159.572} C_VEL
LIN {X 0,Y 390.523,Z 936.091,A -85,B 0,C 180,E1 17156.783,E2 17156.783} C_VEL
LIN {X 0,Y 394.994,Z 918.625,A -85,B 0,C 180,E1 17153.954,E2 17153.954} C_VEL
LIN {X 0,Y 399.347,Z 901.587,A -85,B 0,C 180,E1 17151.597,E2 17151.597} C_VEL
LIN {X 0,Y 403.81,Z 883.52,A -85,B 0,C 180,E1 17149.477,E2 17149.477} C_VEL
LIN {X 0,Y 408.288,Z 864.729,A -85,B 0,C 180,E1 17147.579,E2 17147.579} C_VEL
LIN {X 0,Y 412.725,Z 844.208,A -85,B 0,C 180,E1 17145.852,E2 17145.852} C_VEL
LIN {X 0,Y 416.887,Z 823.456,A -85,B 0,C 180,E1 17144.388,E2 17144.388} C_VEL
LIN {X 0,Y 420.521,Z 802.591,A -85,B 0,C 180,E1 17143.191,E2 17143.191} C_VEL
LIN {X 0,Y 424.071,Z 778.936,A -85,B 0,C 180,E1 17142.11,E2 17142.11} C_VEL
LIN {X 0,Y 426.505,Z 758.787,A -85,B 0,C 180,E1 17141.403,E2 17141.403} C_VEL
LIN {X 0,Y 428.699,Z 733.706,A -85,B 0,C 180,E1 17140.761,E2 17140.761} C_VEL
LIN {X 0,Y 438.036,Z 526.644,A -85,B 0,C 180,E1 17136.831,E2 17136.831} C_VEL
LIN {X 0,Y 440.603,Z 469.683,A -85,B 0,C 180,E1 17135.716,E2 17135.716} C_VEL
LIN {X 0,Y 430.986,Z 454.601,A -85,B 0,C 180,E1 17133.553,E2 17133.553} C_VEL
LIN {X 0,Y 421.638,Z 440.813,A -85,B 0,C 180,E1 17131.287,E2 17131.287} C_VEL
LIN {X 0,Y 412.226,Z 427.545,A -85,B 0,C 180,E1 17128.78,E2 17128.78} C_VEL
LIN {X 0,Y 405.002,Z 417.968,A -85,B 0,C 180,E1 17126.699,E2 17126.699} C_VEL
LIN {X 0,Y 400.612,Z 412.289,A -85,B 0,C 180,E1 17125.342,E2 17125.342} C_VEL
LIN {X 0,Y 396.831,Z 407.628,A -85,B 0,C 180,E1 17124.129,E2 17124.129} C_VEL
LIN {X 0,Y 393.03,Z 402.77,A -85,B 0,C 180,E1 17122.827,E2 17122.827} C_VEL
LIN {X 0,Y 389.846,Z 399.438,A -85,B 0,C 180,E1 17121.713,E2 17121.713} C_VEL
LIN {X 0,Y 388.332,Z 396.969,A -85,B 0,C 180,E1 17121.128,E2 17121.128} C_VEL
LIN {X 0,Y 385.138,Z 394.363,A -85,B 0,C 180,E1 17119.961,E2 17119.961} C_VEL
LIN {X 0,Y 383,Z 390.675,A -85,B 0,C 180,E1 17119.045,E2 17119.045} C_VEL
LIN {X 0,Y 379.763,Z 388.49,A -85,B 0,C 180,E1 17117.782,E2 17117.782} C_VEL
LIN {X 0,Y 377.946,Z 385.476,A -85,B 0,C 180,E1 17116.918,E2 17116.918} C_VEL
LIN {X 0,Y 377.633,Z 384.125,A -85,B 0,C 180,E1 17116.299,E2 17116.299} C_VEL
LIN {X 0,Y 377.617,Z 383.999,A -85,B 0,C 180,E1 17112.333,E2 17112.333} C_VEL
LIN {X 0,Y 377.617,Z 383.995,A -85,B 0,C 180,E1 17108.373,E2 17108.373} C_VEL
LIN {X 0,Y 377.622,Z 384.005,A -85,B 0,C 180,E1 17104.251,E2 17104.251} C_VEL
LIN {X 0,Y 377.623,Z 384.009,A -85,B 0,C 180,E1 17100.151,E2 17100.151} C_VEL
LIN {X 0,Y 377.627,Z 383.998,A -85,B 0,C 180,E1 17096.052,E2 17096.052} C_VEL
LIN {X 0,Y 377.631,Z 383.993,A -85,B 0,C 180,E1 17091.933,E2 17091.933} C_VEL
LIN {X 0,Y 377.634,Z 383.997,A -85,B 0,C 180,E1 17087.926,E2 17087.926} C_VEL
LIN {X 0,Y 377.643,Z 384.003,A -85,B 0,C 180,E1 17083.94,E2 17083.94} C_VEL
LIN {X 0,Y 377.655,Z 384.007,A -85,B 0,C 180,E1 17080.011,E2 17080.011} C_VEL
LIN {X 0,Y 377.669,Z 384,A -85,B 0,C 180,E1 17076.105,E2 17076.105} C_VEL
LIN {X 0,Y 377.679,Z 383.989,A -85,B 0,C 180,E1 17072.057,E2 17072.057} C_VEL
LIN {X 0,Y 377.683,Z 383.989,A -85,B 0,C 180,E1 17068.03,E2 17068.03} C_VEL
LIN {X 0,Y 377.682,Z 383.996,A -85,B 0,C 180,E1 17064.004,E2 17064.004} C_VEL
LIN {X 0,Y 377.695,Z 383.995,A -85,B 0,C 180,E1 17059.902,E2 17059.902} C_VEL
LIN {X 0,Y 377.685,Z 383.988,A -85,B 0,C 180,E1 17055.834,E2 17055.834} C_VEL
LIN {X 0,Y 377.717,Z 384.409,A -85,B 0,C 180,E1 17054.751,E2 17054.751} C_VEL
LIN {X 0,Y 378.207,Z 386.046,A -85,B 0,C 180,E1 17054.238,E2 17054.238} C_VEL
LIN {X 0,Y 380.203,Z 388.897,A -85,B 0,C 180,E1 17053.336,E2 17053.336} C_VEL
LIN {X 0,Y 383.312,Z 391.038,A -85,B 0,C 180,E1 17052.126,E2 17052.126} C_VEL
LIN {X 0,Y 385.385,Z 394.602,A -85,B 0,C 180,E1 17051.258,E2 17051.258} C_VEL
LIN {X 0,Y 388.771,Z 397.509,A -85,B 0,C 180,E1 17050.018,E2 17050.018} C_VEL
LIN {X 0,Y 391.38,Z 401.324,A -85,B 0,C 180,E1 17049.046,E2 17049.046} C_VEL
LIN {X 0,Y 394.09,Z 403.801,A -85,B 0,C 180,E1 17048.138,E2 17048.138} C_VEL
LIN {X 0,Y 397.231,Z 407.976,A -85,B 0,C 180,E1 17047.068,E2 17047.068} C_VEL
LIN {X 0,Y 399.348,Z 410.105,A -85,B 0,C 180,E1 17046.406,E2 17046.406} C_VEL
LIN {X 0,Y 403.102,Z 414.607,A -85,B 0,C 180,E1 17045.246,E2 17045.246} C_VEL
LIN {X 0,Y 409.336,Z 422.523,A -85,B 0,C 180,E1 17043.407,E2 17043.407} C_VEL
LIN {X 0,Y 414.571,Z 429.088,A -85,B 0,C 180,E1 17041.973,E2 17041.973} C_VEL
LIN {X 0,Y 421.76,Z 438.467,A -85,B 0,C 180,E1 17040.122,E2 17040.122} C_VEL
LIN {X 0,Y 431.501,Z 451.665,A -85,B 0,C 180,E1 17037.799,E2 17037.799} C_VEL
LIN {X 0,Y 440.453,Z 464.715,A -85,B 0,C 180,E1 17035.821,E2 17035.821} C_VEL
LIN {X 0,Y 430.918,Z 672.396,A -85,B 0,C 180,E1 17031.888,E2 17031.888} C_VEL
LIN {X 0,Y 428.704,Z 717.579,A -85,B 0,C 180,E1 17031.004,E2 17031.004} C_VEL
LIN {X 0,Y 426.575,Z 740.17,A -85,B 0,C 180,E1 17030.36,E2 17030.36} C_VEL
LIN {X 0,Y 424.81,Z 755.185,A -85,B 0,C 180,E1 17029.809,E2 17029.809} C_VEL
LIN {X 0,Y 423.177,Z 762.649,A -85,B 0,C 180,E1 17029.6,E2 17029.6} C_VEL
LIN {X 0,Y 416.239,Z 781.363,A -85,B 0,C 180,E1 17029.296,E2 17029.296} C_VEL
LIN {X 0,Y 414.276,Z 788.518,A -85,B 0,C 180,E1 17028.993,E2 17028.993} C_VEL
LIN {X 0,Y 410.317,Z 808.994,A -85,B 0,C 180,E1 17027.674,E2 17027.674} C_VEL
LIN {X 0,Y 406.077,Z 828.862,A -85,B 0,C 180,E1 17026.15,E2 17026.15} C_VEL
LIN {X 0,Y 401.396,Z 848.337,A -85,B 0,C 180,E1 17024.345,E2 17024.345} C_VEL
LIN {X 0,Y 396.315,Z 868.239,A -85,B 0,C 180,E1 17022.156,E2 17022.156} C_VEL
LIN {X 0,Y 392.035,Z 884.045,A -85,B 0,C 180,E1 17020.109,E2 17020.109} C_VEL
LIN {X 0,Y 387.066,Z 901.775,A -85,B 0,C 180,E1 17017.416,E2 17017.416} C_VEL
LIN {X 0,Y 382.745,Z 917.322,A -85,B 0,C 180,E1 17014.64,E2 17014.64} C_VEL
LIN {X 0,Y 378.822,Z 931.345,A -85,B 0,C 180,E1 17011.659,E2 17011.659} C_VEL
LIN {X 0,Y 375.476,Z 944.141,A -85,B 0,C 180,E1 17008.47,E2 17008.47} C_VEL
LIN {X 0,Y 372.959,Z 954.561,A -85,B 0,C 180,E1 17005.382,E2 17005.382} C_VEL
LIN {X 0,Y 370.782,Z 964.775,A -85,B 0,C 180,E1 17001.757,E2 17001.757} C_VEL
LIN {X 0,Y 369.498,Z 972.075,A -85,B 0,C 180,E1 16998.603,E2 16998.603} C_VEL
LIN {X 0,Y 368.58,Z 978.773,A -85,B 0,C 180,E1 16994.959,E2 16994.959} C_VEL
LIN {X 0,Y 368.169,Z 983.441,A -85,B 0,C 180,E1 16991.633,E2 16991.633} C_VEL
LIN {X 0,Y 367.965,Z 986.803,A -85,B 0,C 180,E1 16988.14,E2 16988.14} C_VEL
LIN {X 0,Y 367.939,Z 988.542,A -85,B 0,C 180,E1 16985.085,E2 16985.085} C_VEL
LIN {X 0,Y 367.927,Z 989.176,A -85,B 0,C 180,E1 16981.599,E2 16981.599} C_VEL
LIN {X 0,Y 367.936,Z 988.374,A -85,B 0,C 180,E1 16978.363,E2 16978.363} C_VEL
LIN {X 0,Y 368.015,Z 986.185,A -85,B 0,C 180,E1 16974.865,E2 16974.865} C_VEL
LIN {X 0,Y 368.228,Z 982.598,A -85,B 0,C 180,E1 16971.547,E2 16971.547} C_VEL
LIN {X 0,Y 368.76,Z 977.661,A -85,B 0,C 180,E1 16968.159,E2 16968.159} C_VEL
LIN {X 0,Y 369.752,Z 970.849,A -85,B 0,C 180,E1 16964.664,E2 16964.664} C_VEL
LIN {X 0,Y 371.325,Z 962.485,A -85,B 0,C 180,E1 16961.171,E2 16961.171} C_VEL
LIN {X 0,Y 373.52,Z 952.564,A -85,B 0,C 180,E1 16957.807,E2 16957.807} C_VEL
LIN {X 0,Y 376.615,Z 940.313,A -85,B 0,C 180,E1 16954.34,E2 16954.34} C_VEL
LIN {X 0,Y 380.156,Z 927.428,A -85,B 0,C 180,E1 16951.258,E2 16951.258} C_VEL
LIN {X 0,Y 384.143,Z 913.131,A -85,B 0,C 180,E1 16948.382,E2 16948.382} C_VEL
LIN {X 0,Y 388.658,Z 897.547,A -85,B 0,C 180,E1 16945.689,E2 16945.689} C_VEL
LIN {X 0,Y 393.265,Z 881.141,A -85,B 0,C 180,E1 16943.289,E2 16943.289} C_VEL
LIN {X 0,Y 398.558,Z 861.672,A -85,B 0,C 180,E1 16940.87,E2 16940.87} C_VEL
LIN {X 0,Y 403.435,Z 842.815,A -85,B 0,C 180,E1 16938.897,E2 16938.897} C_VEL
LIN {X 0,Y 407.957,Z 823.459,A -85,B 0,C 180,E1 16937.204,E2 16937.204} C_VEL
LIN {X 0,Y 412.338,Z 803.032,A -85,B 0,C 180,E1 16935.698,E2 16935.698} C_VEL
LIN {X 0,Y 416.128,Z 782.279,A -85,B 0,C 180,E1 16934.454,E2 16934.454} C_VEL
LIN {X 0,Y 419.622,Z 760.099,A -85,B 0,C 180,E1 16933.377,E2 16933.377} C_VEL
LIN {X 0,Y 422.323,Z 738.236,A -85,B 0,C 180,E1 16932.564,E2 16932.564} C_VEL
LIN {X 0,Y 424.58,Z 713.386,A -85,B 0,C 180,E1 16931.901,E2 16931.901} C_VEL
LIN {X 0,Y 435.894,Z 500.758,A -85,B 0,C 180,E1 16927.741,E2 16927.741} C_VEL
LIN {X 0,Y 437.682,Z 469.367,A -85,B 0,C 180,E1 16927.12,E2 16927.12} C_VEL
LIN {X 0,Y 430.108,Z 457.717,A -85,B 0,C 180,E1 16925.069,E2 16925.069} C_VEL
LIN {X 0,Y 423.765,Z 448.537,A -85,B 0,C 180,E1 16923.145,E2 16923.145} C_VEL
LIN {X 0,Y 418.043,Z 440.546,A -85,B 0,C 180,E1 16921.177,E2 16921.177} C_VEL
LIN {X 0,Y 414.135,Z 435.355,A -85,B 0,C 180,E1 16919.655,E2 16919.655} C_VEL
LIN {X 0,Y 410.493,Z 430.482,A -85,B 0,C 180,E1 16918.046,E2 16918.046} C_VEL
LIN {X 0,Y 407.127,Z 426.245,A -85,B 0,C 180,E1 16916.34,E2 16916.34} C_VEL
LIN {X 0,Y 406.402,Z 425.059,A -85,B 0,C 180,E1 16915.909,E2 16915.909} C_VEL
LIN {X 0,Y 403.117,Z 421.665,A -85,B 0,C 180,E1 16913.807,E2 16913.807} C_VEL
LIN {X 0,Y 401.848,Z 419.135,A -85,B 0,C 180,E1 16912.71,E2 16912.71} C_VEL
LIN {X 0,Y 398.238,Z 415.923,A -85,B 0,C 180,E1 16907.826,E2 16907.826} C_VEL
LIN {X 0,Y 398.054,Z 415.59,A -85,B 0,C 180,E1 16905.602,E2 16905.602} C_VEL
LIN {X 0,Y 399.383,Z 417.509,A -85,B 0,C 180,E1 16902.217,E2 16902.217} C_VEL
LIN {X 0,Y 402.159,Z 419.577,A -85,B 0,C 180,E1 16899.479,E2 16899.479} C_VEL
LIN {X 0,Y 404.29,Z 423.334,A -85,B 0,C 180,E1 16897.767,E2 16897.767} C_VEL
LIN {X 0,Y 406.806,Z 425.648,A -85,B 0,C 180,E1 16896.306,E2 16896.306} C_VEL
LIN {X 0,Y 409.756,Z 429.864,A -85,B 0,C 180,E1 16894.722,E2 16894.722} C_VEL
LIN {X 0,Y 411.59,Z 432.154,A -85,B 0,C 180,E1 16893.877,E2 16893.877} C_VEL
LIN {X 0,Y 416.804,Z 439.647,A -85,B 0,C 180,E1 16891.693,E2 16891.693} C_VEL
LIN {X 0,Y 422.955,Z 449.208,A -85,B 0,C 180,E1 16889.492,E2 16889.492} C_VEL
LIN {X 0,Y 430.295,Z 461.021,A -85,B 0,C 180,E1 16887.221,E2 16887.221} C_VEL
LIN {X 0,Y 437.652,Z 473.974,A -85,B 0,C 180,E1 16885.198,E2 16885.198} C_VEL
LIN {X 0,Y 427.465,Z 664.156,A -85,B 0,C 180,E1 16881.475,E2 16881.475} C_VEL
LIN {X 0,Y 423.691,Z 736.929,A -85,B 0,C 180,E1 16880.039,E2 16880.039} C_VEL
LIN {X 0,Y 421.25,Z 760.303,A -85,B 0,C 180,E1 16879.394,E2 16879.394} C_VEL
LIN {X 0,Y 418.308,Z 782.279,A -85,B 0,C 180,E1 16878.584,E2 16878.584} C_VEL
LIN {X 0,Y 414.691,Z 803.973,A -85,B 0,C 180,E1 16877.538,E2 16877.538} C_VEL
LIN {X 0,Y 410.325,Z 826.798,A -85,B 0,C 180,E1 16876.164,E2 16876.164} C_VEL
LIN {X 0,Y 405.971,Z 847.082,A -85,B 0,C 180,E1 16874.668,E2 16874.668} C_VEL
LIN {X 0,Y 401.203,Z 867.315,A -85,B 0,C 180,E1 16872.875,E2 16872.875} C_VEL
LIN {X 0,Y 396.612,Z 885.709,A -85,B 0,C 180,E1 16870.958,E2 16870.958} C_VEL
LIN {X 0,Y 391.767,Z 904.007,A -85,B 0,C 180,E1 16868.707,E2 16868.707} C_VEL
LIN {X 0,Y 387.096,Z 921.652,A -85,B 0,C 180,E1 16866.174,E2 16866.174} C_VEL
LIN {X 0,Y 382.753,Z 937.676,A -85,B 0,C 180,E1 16863.453,E2 16863.453} C_VEL
LIN {X 0,Y 378.619,Z 953.618,A -85,B 0,C 180,E1 16860.285,E2 16860.285} C_VEL
LIN {X 0,Y 375.604,Z 965.903,A -85,B 0,C 180,E1 16857.425,E2 16857.425} C_VEL
LIN {X 0,Y 372.838,Z 978.192,A -85,B 0,C 180,E1 16854.06,E2 16854.06} C_VEL
LIN {X 0,Y 370.907,Z 988.136,A -85,B 0,C 180,E1 16850.849,E2 16850.849} C_VEL
LIN {X 0,Y 369.504,Z 996.722,A -85,B 0,C 180,E1 16847.483,E2 16847.483} C_VEL
LIN {X 0,Y 368.663,Z 1003.435,A -85,B 0,C 180,E1 16844.293,E2 16844.293} C_VEL
LIN {X 0,Y 368.17,Z 1009.127,A -85,B 0,C 180,E1 16840.805,E2 16840.805} C_VEL
LIN {X 0,Y 367.982,Z 1012.753,A -85,B 0,C 180,E1 16837.813,E2 16837.813} C_VEL
LIN {X 0,Y 367.924,Z 1015.53,A -85,B 0,C 180,E1 16834.369,E2 16834.369} C_VEL
LIN {X 0,Y 367.923,Z 1016.628,A -85,B 0,C 180,E1 16831.25,E2 16831.25} C_VEL
LIN {X 0,Y 367.927,Z 1016.571,A -85,B 0,C 180,E1 16828.292,E2 16828.292} C_VEL
LIN {X 0,Y 367.929,Z 1015.068,A -85,B 0,C 180,E1 16824.86,E2 16824.86} C_VEL
LIN {X 0,Y 368.017,Z 1012.333,A -85,B 0,C 180,E1 16821.726,E2 16821.726} C_VEL
LIN {X 0,Y 368.26,Z 1007.908,A -85,B 0,C 180,E1 16818.256,E2 16818.256} C_VEL
LIN {X 0,Y 368.839,Z 1002.035,A -85,B 0,C 180,E1 16814.921,E2 16814.921} C_VEL
LIN {X 0,Y 369.869,Z 994.738,A -85,B 0,C 180,E1 16811.567,E2 16811.567} C_VEL
LIN {X 0,Y 371.453,Z 985.603,A -85,B 0,C 180,E1 16808.2,E2 16808.2} C_VEL
LIN {X 0,Y 373.727,Z 974.762,A -85,B 0,C 180,E1 16804.831,E2 16804.831} C_VEL
LIN {X 0,Y 376.432,Z 963.113,A -85,B 0,C 180,E1 16801.791,E2 16801.791} C_VEL
LIN {X 0,Y 380.232,Z 948.085,A -85,B 0,C 180,E1 16798.454,E2 16798.454} C_VEL
LIN {X 0,Y 384.25,Z 933.113,A -85,B 0,C 180,E1 16795.629,E2 16795.629} C_VEL
LIN {X 0,Y 388.643,Z 916.654,A -85,B 0,C 180,E1 16792.993,E2 16792.993} C_VEL
LIN {X 0,Y 393.419,Z 898.962,A -85,B 0,C 180,E1 16790.561,E2 16790.561} C_VEL
LIN {X 0,Y 398.034,Z 880.935,A -85,B 0,C 180,E1 16788.466,E2 16788.466} C_VEL
LIN {X 0,Y 403.128,Z 859.991,A -85,B 0,C 180,E1 16786.404,E2 16786.404} C_VEL
LIN {X 0,Y 407.426,Z 840.969,A -85,B 0,C 180,E1 16784.836,E2 16784.836} C_VEL
LIN {X 0,Y 411.8,Z 819.473,A -85,B 0,C 180,E1 16783.367,E2 16783.367} C_VEL
LIN {X 0,Y 415.347,Z 799.734,A -85,B 0,C 180,E1 16782.257,E2 16782.257} C_VEL
LIN {X 0,Y 418.802,Z 776.823,A -85,B 0,C 180,E1 16781.235,E2 16781.235} C_VEL
LIN {X 0,Y 421.31,Z 756.598,A -85,B 0,C 180,E1 16780.539,E2 16780.539} C_VEL
LIN {X 0,Y 423.394,Z 732.585,A -85,B 0,C 180,E1 16779.936,E2 16779.936} C_VEL
LIN {X 0,Y 433.274,Z 523.725,A -85,B 0,C 180,E1 16775.939,E2 16775.939} C_VEL
LIN {X 0,Y 435.628,Z 473.714,A -85,B 0,C 180,E1 16774.957,E2 16774.957} C_VEL
LIN {X 0,Y 425.509,Z 457.746,A -85,B 0,C 180,E1 16772.594,E2 16772.594} C_VEL
LIN {X 0,Y 416.281,Z 444.128,A -85,B 0,C 180,E1 16770.251,E2 16770.251} C_VEL
LIN {X 0,Y 406.213,Z 430.014,A -85,B 0,C 180,E1 16767.445,E2 16767.445} C_VEL
LIN {X 0,Y 398.009,Z 419.278,A -85,B 0,C 180,E1 16764.923,E2 16764.923} C_VEL
LIN {X 0,Y 394.085,Z 414.423,A -85,B 0,C 180,E1 16763.632,E2 16763.632} C_VEL
LIN {X 0,Y 390.628,Z 409.986,A -85,B 0,C 180,E1 16762.419,E2 16762.419} C_VEL
LIN {X 0,Y 387.3,Z 406.271,A -85,B 0,C 180,E1 16761.227,E2 16761.227} C_VEL
LIN {X 0,Y 385.966,Z 404.299,A -85,B 0,C 180,E1 16760.707,E2 16760.707} C_VEL
LIN {X 0,Y 382.682,Z 401.238,A -85,B 0,C 180,E1 16759.458,E2 16759.458} C_VEL
LIN {X 0,Y 380.871,Z 398.182,A -85,B 0,C 180,E1 16758.679,E2 16758.679} C_VEL
LIN {X 0,Y 377.712,Z 395.814,A -85,B 0,C 180,E1 16757.405,E2 16757.405} C_VEL
LIN {X 0,Y 375.592,Z 392.312,A -85,B 0,C 180,E1 16756.39,E2 16756.39} C_VEL
LIN {X 0,Y 373.936,Z 391.081,A -85,B 0,C 180,E1 16755.667,E2 16755.667} C_VEL
LIN {X 0,Y 371.123,Z 388.675,A -85,B 0,C 180,E1 16754.35,E2 16754.35} C_VEL
LIN {X 0,Y 369.847,Z 385.709,A -85,B 0,C 180,E1 16753.443,E2 16753.443} C_VEL
LIN {X 0,Y 369.683,Z 385.019,A -85,B 0,C 180,E1 16752.654,E2 16752.654} C_VEL
LIN {X 0,Y 369.681,Z 384.983,A -85,B 0,C 180,E1 16748.554,E2 16748.554} C_VEL
LIN {X 0,Y 369.693,Z 384.986,A -85,B 0,C 180,E1 16744.653,E2 16744.653} C_VEL
LIN {X 0,Y 369.702,Z 384.997,A -85,B 0,C 180,E1 16740.619,E2 16740.619} C_VEL
LIN {X 0,Y 369.708,Z 384.99,A -85,B 0,C 180,E1 16736.588,E2 16736.588} C_VEL
LIN {X 0,Y 369.716,Z 384.981,A -85,B 0,C 180,E1 16732.541,E2 16732.541} C_VEL
LIN {X 0,Y 369.72,Z 384.979,A -85,B 0,C 180,E1 16728.455,E2 16728.455} C_VEL
LIN {X 0,Y 369.735,Z 384.981,A -85,B 0,C 180,E1 16724.471,E2 16724.471} C_VEL
LIN {X 0,Y 369.738,Z 384.987,A -85,B 0,C 180,E1 16720.407,E2 16720.407} C_VEL
LIN {X 0,Y 369.747,Z 384.991,A -85,B 0,C 180,E1 16716.408,E2 16716.408} C_VEL
LIN {X 0,Y 369.747,Z 384.979,A -85,B 0,C 180,E1 16712.281,E2 16712.281} C_VEL
LIN {X 0,Y 369.747,Z 384.977,A -85,B 0,C 180,E1 16708.175,E2 16708.175} C_VEL
LIN {X 0,Y 369.744,Z 384.983,A -85,B 0,C 180,E1 16704.068,E2 16704.068} C_VEL
LIN {X 0,Y 369.756,Z 384.984,A -85,B 0,C 180,E1 16699.92,E2 16699.92} C_VEL
LIN {X 0,Y 369.787,Z 385.274,A -85,B 0,C 180,E1 16698.097,E2 16698.097} C_VEL
LIN {X 0,Y 370.144,Z 386.705,A -85,B 0,C 180,E1 16697.505,E2 16697.505} C_VEL
LIN {X 0,Y 371.825,Z 389.47,A -85,B 0,C 180,E1 16696.591,E2 16696.591} C_VEL
LIN {X 0,Y 375.561,Z 392.206,A -85,B 0,C 180,E1 16694.913,E2 16694.913} C_VEL
LIN {X 0,Y 377.643,Z 395.69,A -85,B 0,C 180,E1 16693.932,E2 16693.932} C_VEL
LIN {X 0,Y 381.134,Z 398.553,A -85,B 0,C 180,E1 16692.508,E2 16692.508} C_VEL
LIN {X 0,Y 383.653,Z 402.373,A -85,B 0,C 180,E1 16691.461,E2 16691.461} C_VEL
LIN {X 0,Y 386.558,Z 404.975,A -85,B 0,C 180,E1 16690.381,E2 16690.381} C_VEL
LIN {X 0,Y 389.591,Z 409.061,A -85,B 0,C 180,E1 16689.247,E2 16689.247} C_VEL
LIN {X 0,Y 391.767,Z 411.138,A -85,B 0,C 180,E1 16688.508,E2 16688.508} C_VEL
LIN {X 0,Y 395.294,Z 415.603,A -85,B 0,C 180,E1 16687.297,E2 16687.297} C_VEL
LIN {X 0,Y 397.046,Z 417.547,A -85,B 0,C 180,E1 16686.732,E2 16686.732} C_VEL
LIN {X 0,Y 401.951,Z 423.591,A -85,B 0,C 180,E1 16685.199,E2 16685.199} C_VEL
LIN {X 0,Y 406.921,Z 429.89,A -85,B 0,C 180,E1 16683.726,E2 16683.726} C_VEL
LIN {X 0,Y 413.867,Z 438.603,A -85,B 0,C 180,E1 16681.81,E2 16681.81} C_VEL
LIN {X 0,Y 425.337,Z 454.179,A -85,B 0,C 180,E1 16678.911,E2 16678.911} C_VEL
LIN {X 0,Y 435.44,Z 468.713,A -85,B 0,C 180,E1 16676.589,E2 16676.589} C_VEL
LIN {X 0,Y 425.74,Z 671.1,A -85,B 0,C 180,E1 16672.726,E2 16672.726} C_VEL
LIN {X 0,Y 423.355,Z 717.83,A -85,B 0,C 180,E1 16671.805,E2 16671.805} C_VEL
LIN {X 0,Y 421.137,Z 740.584,A -85,B 0,C 180,E1 16671.153,E2 16671.153} C_VEL
LIN {X 0,Y 418.075,Z 764.632,A -85,B 0,C 180,E1 16670.212,E2 16670.212} C_VEL
LIN {X 0,Y 414.897,Z 784.693,A -85,B 0,C 180,E1 16669.205,E2 16669.205} C_VEL
LIN {X 0,Y 414.276,Z 788.518,A -85,B 0,C 180,E1 16668.993,E2 16668.993} C_VEL
LIN {X 0,Y 412.229,Z 795.659,A -85,B 0,C 180,E1 16668.663,E2 16668.663} C_VEL
LIN {X 0,Y 404.333,Z 813.698,A -85,B 0,C 180,E1 16668.063,E2 16668.063} C_VEL
LIN {X 0,Y 402.128,Z 820.441,A -85,B 0,C 180,E1 16667.644,E2 16667.644} C_VEL
LIN {X 0,Y 397.563,Z 839.865,A -85,B 0,C 180,E1 16665.98,E2 16665.98} C_VEL
LIN {X 0,Y 392.53,Z 859.155,A -85,B 0,C 180,E1 16663.999,E2 16663.999} C_VEL
LIN {X 0,Y 387.586,Z 877.171,A -85,B 0,C 180,E1 16661.83,E2 16661.83} C_VEL
LIN {X 0,Y 382.779,Z 893.676,A -85,B 0,C 180,E1 16659.467,E2 16659.467} C_VEL
LIN {X 0,Y 378.14,Z 909.504,A -85,B 0,C 180,E1 16656.829,E2 16656.829} C_VEL
LIN {X 0,Y 373.865,Z 923.858,A -85,B 0,C 180,E1 16654.008,E2 16654.008} C_VEL
LIN {X 0,Y 369.858,Z 937.839,A -85,B 0,C 180,E1 16650.77,E2 16650.77} C_VEL
LIN {X 0,Y 366.802,Z 949.236,A -85,B 0,C 180,E1 16647.652,E2 16647.652} C_VEL
LIN {X 0,Y 364.183,Z 959.852,A -85,B 0,C 180,E1 16644.165,E2 16644.165} C_VEL
LIN {X 0,Y 362.319,Z 968.84,A -85,B 0,C 180,E1 16640.625,E2 16640.625} C_VEL
LIN {X 0,Y 361.095,Z 975.967,A -85,B 0,C 180,E1 16637.081,E2 16637.081} C_VEL
LIN {X 0,Y 360.362,Z 981.803,A -85,B 0,C 180,E1 16633.39,E2 16633.39} C_VEL
LIN {X 0,Y 360.067,Z 985.454,A -85,B 0,C 180,E1 16630.193,E2 16630.193} C_VEL
LIN {X 0,Y 359.944,Z 988.15,A -85,B 0,C 180,E1 16626.764,E2 16626.764} C_VEL
LIN {X 0,Y 359.923,Z 989.313,A -85,B 0,C 180,E1 16623.428,E2 16623.428} C_VEL
LIN {X 0,Y 359.92,Z 989.312,A -85,B 0,C 180,E1 16620.36,E2 16620.36} C_VEL
LIN {X 0,Y 359.96,Z 987.972,A -85,B 0,C 180,E1 16616.82,E2 16616.82} C_VEL
LIN {X 0,Y 360.071,Z 985.462,A -85,B 0,C 180,E1 16613.639,E2 16613.639} C_VEL
LIN {X 0,Y 360.436,Z 981.452,A -85,B 0,C 180,E1 16610.144,E2 16610.144} C_VEL
LIN {X 0,Y 361.162,Z 975.784,A -85,B 0,C 180,E1 16606.636,E2 16606.636} C_VEL
LIN {X 0,Y 362.453,Z 968.463,A -85,B 0,C 180,E1 16603.023,E2 16603.023} C_VEL
LIN {X 0,Y 364.35,Z 959.58,A -85,B 0,C 180,E1 16599.54,E2 16599.54} C_VEL
LIN {X 0,Y 367.232,Z 948.133,A -85,B 0,C 180,E1 16595.83,E2 16595.83} C_VEL
LIN {X 0,Y 370.519,Z 936.404,A -85,B 0,C 180,E1 16592.649,E2 16592.649} C_VEL
LIN {X 0,Y 374.394,Z 923.07,A -85,B 0,C 180,E1 16589.609,E2 16589.609} C_VEL
LIN {X 0,Y 378.857,Z 908.485,A -85,B 0,C 180,E1 16586.759,E2 16586.759} C_VEL
LIN {X 0,Y 383.693,Z 892.244,A -85,B 0,C 180,E1 16584.082,E2 16584.082} C_VEL
LIN {X 0,Y 389.203,Z 873.519,A -85,B 0,C 180,E1 16581.475,E2 16581.475} C_VEL
LIN {X 0,Y 394.122,Z 856.039,A -85,B 0,C 180,E1 16579.411,E2 16579.411} C_VEL
LIN {X 0,Y 399.112,Z 836.749,A -85,B 0,C 180,E1 16577.496,E2 16577.496} C_VEL
LIN {X 0,Y 403.994,Z 816.452,A -85,B 0,C 180,E1 16575.798,E2 16575.798} C_VEL
LIN {X 0,Y 408.289,Z 795.916,A -85,B 0,C 180,E1 16574.393,E2 16574.393} C_VEL
LIN {X 0,Y 412.272,Z 774.249,A -85,B 0,C 180,E1 16573.178,E2 16573.178} C_VEL
LIN {X 0,Y 415.373,Z 753.63,A -85,B 0,C 180,E1 16572.262,E2 16572.262} C_VEL
LIN {X 0,Y 418.203,Z 729.949,A -85,B 0,C 180,E1 16571.459,E2 16571.459} C_VEL
LIN {X 0,Y 419.959,Z 708.435,A -85,B 0,C 180,E1 16570.937,E2 16570.937} C_VEL
LIN {X 0,Y 431.422,Z 502.905,A -85,B 0,C 180,E1 16566.891,E2 16566.891} C_VEL
LIN {X 0,Y 433.139,Z 473.589,A -85,B 0,C 180,E1 16566.296,E2 16566.296} C_VEL
LIN {X 0,Y 425.326,Z 461.45,A -85,B 0,C 180,E1 16564.045,E2 16564.045} C_VEL
LIN {X 0,Y 418.734,Z 451.921,A -85,B 0,C 180,E1 16561.882,E2 16561.882} C_VEL
LIN {X 0,Y 415.043,Z 446.804,A -85,B 0,C 180,E1 16560.515,E2 16560.515} C_VEL
LIN {X 0,Y 411.989,Z 442.582,A -85,B 0,C 180,E1 16559.27,E2 16559.27} C_VEL
LIN {X 0,Y 408.567,Z 437.881,A -85,B 0,C 180,E1 16557.686,E2 16557.686} C_VEL
LIN {X 0,Y 405.216,Z 433.366,A -85,B 0,C 180,E1 16555.897,E2 16555.897} C_VEL
LIN {X 0,Y 403.31,Z 431.459,A -85,B 0,C 180,E1 16554.738,E2 16554.738} C_VEL
LIN {X 0,Y 400.834,Z 427.68,A -85,B 0,C 180,E1 16552.836,E2 16552.836} C_VEL
LIN {X 0,Y 400.376,Z 426.884,A -85,B 0,C 180,E1 16552.395,E2 16552.395} C_VEL
LIN {X 0,Y 397.109,Z 423.79,A -85,B 0,C 180,E1 16547.643,E2 16547.643} C_VEL
LIN {X 0,Y 396.977,Z 423.53,A -85,B 0,C 180,E1 16545.562,E2 16545.562} C_VEL
LIN {X 0,Y 398.441,Z 425.629,A -85,B 0,C 180,E1 16542.01,E2 16542.01} C_VEL
LIN {X 0,Y 400.751,Z 427.373,A -85,B 0,C 180,E1 16539.709,E2 16539.709} C_VEL
LIN {X 0,Y 402.941,Z 431.158,A -85,B 0,C 180,E1 16537.919,E2 16537.919} C_VEL
LIN {X 0,Y 405.147,Z 433.274,A -85,B 0,C 180,E1 16536.589,E2 16536.589} C_VEL
LIN {X 0,Y 408.169,Z 437.572,A -85,B 0,C 180,E1 16534.927,E2 16534.927} C_VEL
LIN {X 0,Y 411.605,Z 442.316,A -85,B 0,C 180,E1 16533.335,E2 16533.335} C_VEL
LIN {X 0,Y 417.599,Z 451.522,A -85,B 0,C 180,E1 16530.92,E2 16530.92} C_VEL
LIN {X 0,Y 424.915,Z 463.514,A -85,B 0,C 180,E1 16528.429,E2 16528.429} C_VEL
LIN {X 0,Y 432.307,Z 476.448,A -85,B 0,C 180,E1 16526.244,E2 16526.244} C_VEL
LIN {X 0,Y 433.116,Z 478.209,A -85,B 0,C 180,E1 16526.009,E2 16526.009} C_VEL
LIN {X 0,Y 422.412,Z 668.051,A -85,B 0,C 180,E1 16522.261,E2 16522.261} C_VEL
LIN {X 0,Y 418.648,Z 736.809,A -85,B 0,C 180,E1 16520.891,E2 16520.891} C_VEL
LIN {X 0,Y 416.12,Z 760.014,A -85,B 0,C 180,E1 16520.246,E2 16520.246} C_VEL
LIN {X 0,Y 413.026,Z 782.098,A -85,B 0,C 180,E1 16519.427,E2 16519.427} C_VEL
LIN {X 0,Y 409.28,Z 803.68,A -85,B 0,C 180,E1 16518.382,E2 16518.382} C_VEL
LIN {X 0,Y 404.776,Z 826.254,A -85,B 0,C 180,E1 16517.019,E2 16517.019} C_VEL
LIN {X 0,Y 400.19,Z 846.636,A -85,B 0,C 180,E1 16515.509,E2 16515.509} C_VEL
LIN {X 0,Y 395.175,Z 866.999,A -85,B 0,C 180,E1 16513.692,E2 16513.692} C_VEL
LIN {X 0,Y 390.37,Z 885.359,A -85,B 0,C 180,E1 16511.758,E2 16511.758} C_VEL
LIN {X 0,Y 385.18,Z 904.021,A -85,B 0,C 180,E1 16509.433,E2 16509.433} C_VEL
LIN {X 0,Y 380.441,Z 920.972,A -85,B 0,C 180,E1 16506.97,E2 16506.97} C_VEL
LIN {X 0,Y 376.022,Z 936.438,A -85,B 0,C 180,E1 16504.317,E2 16504.317} C_VEL
LIN {X 0,Y 372.002,Z 951.041,A -85,B 0,C 180,E1 16501.432,E2 16501.432} C_VEL
LIN {X 0,Y 368.505,Z 964.227,A -85,B 0,C 180,E1 16498.352,E2 16498.352} C_VEL
LIN {X 0,Y 365.483,Z 976.769,A -85,B 0,C 180,E1 16494.921,E2 16494.921} C_VEL
LIN {X 0,Y 363.337,Z 986.833,A -85,B 0,C 180,E1 16491.643,E2 16491.643} C_VEL
LIN {X 0,Y 361.688,Z 996.058,A -85,B 0,C 180,E1 16488.02,E2 16488.02} C_VEL
LIN {X 0,Y 360.76,Z 1002.787,A -85,B 0,C 180,E1 16484.777,E2 16484.777} C_VEL
LIN {X 0,Y 360.192,Z 1008.808,A -85,B 0,C 180,E1 16481.047,E2 16481.047} C_VEL
LIN {X 0,Y 360.001,Z 1012.44,A -85,B 0,C 180,E1 16477.987,E2 16477.987} C_VEL
LIN {X 0,Y 359.927,Z 1015.224,A -85,B 0,C 180,E1 16474.466,E2 16474.466} C_VEL
LIN {X 0,Y 359.929,Z 1016.328,A -85,B 0,C 180,E1 16471.278,E2 16471.278} C_VEL
LIN {X 0,Y 359.932,Z 1016.273,A -85,B 0,C 180,E1 16468.254,E2 16468.254} C_VEL
LIN {X 0,Y 359.933,Z 1014.769,A -85,B 0,C 180,E1 16464.745,E2 16464.745} C_VEL
LIN {X 0,Y 360.025,Z 1012.034,A -85,B 0,C 180,E1 16461.541,E2 16461.541} C_VEL
LIN {X 0,Y 360.295,Z 1007.605,A -85,B 0,C 180,E1 16457.992,E2 16457.992} C_VEL
LIN {X 0,Y 360.924,Z 1001.728,A -85,B 0,C 180,E1 16454.582,E2 16454.582} C_VEL
LIN {X 0,Y 362.033,Z 994.422,A -85,B 0,C 180,E1 16451.154,E2 16451.154} C_VEL
LIN {X 0,Y 363.727,Z 985.276,A -85,B 0,C 180,E1 16447.713,E2 16447.713} C_VEL
LIN {X 0,Y 366.162,Z 974.423,A -85,B 0,C 180,E1 16444.274,E2 16444.274} C_VEL
LIN {X 0,Y 369.06,Z 962.762,A -85,B 0,C 180,E1 16441.175,E2 16441.175} C_VEL
LIN {X 0,Y 373.098,Z 947.699,A -85,B 0,C 180,E1 16437.778,E2 16437.778} C_VEL
LIN {X 0,Y 377.339,Z 932.716,A -85,B 0,C 180,E1 16434.908,E2 16434.908} C_VEL
LIN {X 0,Y 381.996,Z 916.175,A -85,B 0,C 180,E1 16432.229,E2 16432.229} C_VEL
LIN {X 0,Y 386.99,Z 898.473,A -85,B 0,C 180,E1 16429.773,E2 16429.773} C_VEL
LIN {X 0,Y 391.824,Z 880.42,A -85,B 0,C 180,E1 16427.657,E2 16427.657} C_VEL
LIN {X 0,Y 397.136,Z 859.535,A -85,B 0,C 180,E1 16425.588,E2 16425.588} C_VEL
LIN {X 0,Y 401.71,Z 840.103,A -85,B 0,C 180,E1 16423.981,E2 16423.981} C_VEL
LIN {X 0,Y 406.218,Z 818.622,A -85,B 0,C 180,E1 16422.517,E2 16422.517} C_VEL
LIN {X 0,Y 409.905,Z 798.784,A -85,B 0,C 180,E1 16421.402,E2 16421.402} C_VEL
LIN {X 0,Y 413.413,Z 776.175,A -85,B 0,C 180,E1 16420.397,E2 16420.397} C_VEL
LIN {X 0,Y 416.061,Z 755.55,A -85,B 0,C 180,E1 16419.691,E2 16419.691} C_VEL
LIN {X 0,Y 418.157,Z 731.776,A -85,B 0,C 180,E1 16419.098,E2 16419.098} C_VEL
LIN {X 0,Y 428.391,Z 524.281,A -85,B 0,C 180,E1 16415.099,E2 16415.099} C_VEL
LIN {X 0,Y 430.701,Z 477.757,A -85,B 0,C 180,E1 16414.179,E2 16414.179} C_VEL
LIN {X 0,Y 420.711,Z 461.966,A -85,B 0,C 180,E1 16411.763,E2 16411.763} C_VEL
LIN {X 0,Y 411.9,Z 448.868,A -85,B 0,C 180,E1 16409.442,E2 16409.442} C_VEL
LIN {X 0,Y 402.893,Z 436.177,A -85,B 0,C 180,E1 16406.85,E2 16406.85} C_VEL
LIN {X 0,Y 395.224,Z 426.017,A -85,B 0,C 180,E1 16404.432,E2 16404.432} C_VEL
LIN {X 0,Y 388.423,Z 417.339,A -85,B 0,C 180,E1 16402.075,E2 16402.075} C_VEL
LIN {X 0,Y 384.87,Z 413.242,A -85,B 0,C 180,E1 16400.769,E2 16400.769} C_VEL
LIN {X 0,Y 383.627,Z 411.586,A -85,B 0,C 180,E1 16400.281,E2 16400.281} C_VEL
LIN {X 0,Y 380.228,Z 408.093,A -85,B 0,C 180,E1 16398.95,E2 16398.95} C_VEL
LIN {X 0,Y 378.578,Z 405.575,A -85,B 0,C 180,E1 16398.238,E2 16398.238} C_VEL
LIN {X 0,Y 375.28,Z 402.646,A -85,B 0,C 180,E1 16396.842,E2 16396.842} C_VEL
LIN {X 0,Y 373.245,Z 399.291,A -85,B 0,C 180,E1 16395.857,E2 16395.857} C_VEL
LIN {X 0,Y 369.751,Z 396.729,A -85,B 0,C 180,E1 16394.245,E2 16394.245} C_VEL
LIN {X 0,Y 367.877,Z 393.436,A -85,B 0,C 180,E1 16393.197,E2 16393.197} C_VEL
LIN {X 0,Y 366.705,Z 392.439,A -85,B 0,C 180,E1 16392.598,E2 16392.598} C_VEL
LIN {X 0,Y 363.371,Z 389.901,A -85,B 0,C 180,E1 16390.784,E2 16390.784} C_VEL
LIN {X 0,Y 361.874,Z 386.579,A -85,B 0,C 180,E1 16389.542,E2 16389.542} C_VEL
LIN {X 0,Y 361.747,Z 385.995,A -85,B 0,C 180,E1 16388.583,E2 16388.583} C_VEL
LIN {X 0,Y 361.751,Z 385.975,A -85,B 0,C 180,E1 16384.597,E2 16384.597} C_VEL
LIN {X 0,Y 361.757,Z 385.988,A -85,B 0,C 180,E1 16380.474,E2 16380.474} C_VEL
LIN {X 0,Y 361.758,Z 385.977,A -85,B 0,C 180,E1 16376.355,E2 16376.355} C_VEL
LIN {X 0,Y 361.76,Z 385.97,A -85,B 0,C 180,E1 16372.216,E2 16372.216} C_VEL
LIN {X 0,Y 361.766,Z 385.97,A -85,B 0,C 180,E1 16368.198,E2 16368.198} C_VEL
LIN {X 0,Y 361.773,Z 385.976,A -85,B 0,C 180,E1 16364.12,E2 16364.12} C_VEL
LIN {X 0,Y 361.776,Z 385.985,A -85,B 0,C 180,E1 16359.977,E2 16359.977} C_VEL
LIN {X 0,Y 361.786,Z 385.976,A -85,B 0,C 180,E1 16356.029,E2 16356.029} C_VEL
LIN {X 0,Y 361.795,Z 385.967,A -85,B 0,C 180,E1 16351.977,E2 16351.977} C_VEL
LIN {X 0,Y 361.801,Z 385.966,A -85,B 0,C 180,E1 16347.953,E2 16347.953} C_VEL
LIN {X 0,Y 361.796,Z 385.977,A -85,B 0,C 180,E1 16343.79,E2 16343.79} C_VEL
LIN {X 0,Y 361.858,Z 386.283,A -85,B 0,C 180,E1 16341.941,E2 16341.941} C_VEL
LIN {X 0,Y 362.234,Z 387.814,A -85,B 0,C 180,E1 16341.239,E2 16341.239} C_VEL
LIN {X 0,Y 364.039,Z 390.589,A -85,B 0,C 180,E1 16340.109,E2 16340.109} C_VEL
LIN {X 0,Y 367.756,Z 393.168,A -85,B 0,C 180,E1 16338.145,E2 16338.145} C_VEL
LIN {X 0,Y 369.665,Z 396.574,A -85,B 0,C 180,E1 16337.095,E2 16337.095} C_VEL
LIN {X 0,Y 372.891,Z 399.085,A -85,B 0,C 180,E1 16335.585,E2 16335.585} C_VEL
LIN {X 0,Y 373.593,Z 399.845,A -85,B 0,C 180,E1 16335.26,E2 16335.26} C_VEL
LIN {X 0,Y 376.038,Z 403.511,A -85,B 0,C 180,E1 16334.117,E2 16334.117} C_VEL
LIN {X 0,Y 379.102,Z 406.181,A -85,B 0,C 180,E1 16332.843,E2 16332.843} C_VEL
LIN {X 0,Y 382.049,Z 410.235,A -85,B 0,C 180,E1 16331.619,E2 16331.619} C_VEL
LIN {X 0,Y 384.344,Z 412.333,A -85,B 0,C 180,E1 16330.758,E2 16330.758} C_VEL
LIN {X 0,Y 387.698,Z 416.68,A -85,B 0,C 180,E1 16329.487,E2 16329.487} C_VEL
LIN {X 0,Y 389.569,Z 418.64,A -85,B 0,C 180,E1 16328.834,E2 16328.834} C_VEL
LIN {X 0,Y 393.365,Z 423.222,A -85,B 0,C 180,E1 16327.528,E2 16327.528} C_VEL
LIN {X 0,Y 399.478,Z 430.8,A -85,B 0,C 180,E1 16325.565,E2 16325.565} C_VEL
LIN {X 0,Y 407.704,Z 441.2,A -85,B 0,C 180,E1 16323.135,E2 16323.135} C_VEL
LIN {X 0,Y 418.667,Z 455.889,A -85,B 0,C 180,E1 16320.21,E2 16320.21} C_VEL
LIN {X 0,Y 430.513,Z 472.84,A -85,B 0,C 180,E1 16317.367,E2 16317.367} C_VEL
LIN {X 0,Y 420.138,Z 680.398,A -85,B 0,C 180,E1 16313.38,E2 16313.38} C_VEL
LIN {X 0,Y 418.002,Z 718.929,A -85,B 0,C 180,E1 16312.603,E2 16312.603} C_VEL
LIN {X 0,Y 415.736,Z 741.284,A -85,B 0,C 180,E1 16311.956,E2 16311.956} C_VEL
LIN {X 0,Y 412.569,Z 765.146,A -85,B 0,C 180,E1 16311.014,E2 16311.014} C_VEL
LIN {X 0,Y 409.259,Z 785.279,A -85,B 0,C 180,E1 16309.995,E2 16309.995} C_VEL
LIN {X 0,Y 405.062,Z 806.963,A -85,B 0,C 180,E1 16308.637,E2 16308.637} C_VEL
LIN {X 0,Y 402.128,Z 820.441,A -85,B 0,C 180,E1 16307.644,E2 16307.644} C_VEL
LIN {X 0,Y 399.859,Z 827.375,A -85,B 0,C 180,E1 16307.194,E2 16307.194} C_VEL
LIN {X 0,Y 391.224,Z 844.343,A -85,B 0,C 180,E1 16306.277,E2 16306.277} C_VEL
LIN {X 0,Y 388.809,Z 850.617,A -85,B 0,C 180,E1 16305.746,E2 16305.746} C_VEL
LIN {X 0,Y 383.427,Z 869.797,A -85,B 0,C 180,E1 16303.568,E2 16303.568} C_VEL
LIN {X 0,Y 378.374,Z 886.957,A -85,B 0,C 180,E1 16301.271,E2 16301.271} C_VEL
LIN {X 0,Y 373.473,Z 902.755,A -85,B 0,C 180,E1 16298.773,E2 16298.773} C_VEL
LIN {X 0,Y 368.689,Z 918.291,A -85,B 0,C 180,E1 16295.91,E2 16295.91} C_VEL
LIN {X 0,Y 364.417,Z 932.001,A -85,B 0,C 180,E1 16292.894,E2 16292.894} C_VEL
LIN {X 0,Y 360.597,Z 945.036,A -85,B 0,C 180,E1 16289.519,E2 16289.519} C_VEL
LIN {X 0,Y 357.714,Z 955.587,A -85,B 0,C 180,E1 16286.262,E2 16286.262} C_VEL
LIN {X 0,Y 355.289,Z 965.538,A -85,B 0,C 180,E1 16282.557,E2 16282.557} C_VEL
LIN {X 0,Y 353.737,Z 973.212,A -85,B 0,C 180,E1 16279.079,E2 16279.079} C_VEL
LIN {X 0,Y 352.742,Z 979.344,A -85,B 0,C 180,E1 16275.551,E2 16275.551} C_VEL
LIN {X 0,Y 352.246,Z 983.934,A -85,B 0,C 180,E1 16272.143,E2 16272.143} C_VEL
LIN {X 0,Y 352.01,Z 987.336,A -85,B 0,C 180,E1 16268.501,E2 16268.501} C_VEL
LIN {X 0,Y 351.953,Z 989.101,A -85,B 0,C 180,E1 16265.312,E2 16265.312} C_VEL
LIN {X 0,Y 351.939,Z 989.788,A -85,B 0,C 180,E1 16261.672,E2 16261.672} C_VEL
LIN {X 0,Y 351.951,Z 989.015,A -85,B 0,C 180,E1 16258.289,E2 16258.289} C_VEL
LIN {X 0,Y 352.041,Z 986.999,A -85,B 0,C 180,E1 16254.787,E2 16254.787} C_VEL
LIN {X 0,Y 352.314,Z 983.311,A -85,B 0,C 180,E1 16251.152,E2 16251.152} C_VEL
LIN {X 0,Y 352.958,Z 978.391,A -85,B 0,C 180,E1 16247.603,E2 16247.603} C_VEL
LIN {X 0,Y 354.108,Z 971.601,A -85,B 0,C 180,E1 16243.939,E2 16243.939} C_VEL
LIN {X 0,Y 355.969,Z 963.146,A -85,B 0,C 180,E1 16240.244,E2 16240.244} C_VEL
LIN {X 0,Y 358.432,Z 953.442,A -85,B 0,C 180,E1 16236.808,E2 16236.808} C_VEL
LIN {X 0,Y 361.985,Z 941.072,A -85,B 0,C 180,E1 16233.156,E2 16233.156} C_VEL
LIN {X 0,Y 365.836,Z 928.649,A -85,B 0,C 180,E1 16230.07,E2 16230.07} C_VEL
LIN {X 0,Y 370.407,Z 914.076,A -85,B 0,C 180,E1 16227.022,E2 16227.022} C_VEL
LIN {X 0,Y 375.483,Z 898.292,A -85,B 0,C 180,E1 16224.211,E2 16224.211} C_VEL
LIN {X 0,Y 380.579,Z 881.868,A -85,B 0,C 180,E1 16221.743,E2 16221.743} C_VEL
LIN {X 0,Y 386.215,Z 863.095,A -85,B 0,C 180,E1 16219.353,E2 16219.353} C_VEL
LIN {X 0,Y 391.379,Z 844.827,A -85,B 0,C 180,E1 16217.392,E2 16217.392} C_VEL
LIN {X 0,Y 396.543,Z 824.722,A -85,B 0,C 180,E1 16215.586,E2 16215.586} C_VEL
LIN {X 0,Y 401.295,Z 804.403,A -85,B 0,C 180,E1 16214.06,E2 16214.06} C_VEL
LIN {X 0,Y 405.597,Z 782.796,A -85,B 0,C 180,E1 16212.747,E2 16212.747} C_VEL
LIN {X 0,Y 409.453,Z 760.031,A -85,B 0,C 180,E1 16211.639,E2 16211.639} C_VEL
LIN {X 0,Y 412.355,Z 738.284,A -85,B 0,C 180,E1 16210.829,E2 16210.829} C_VEL
LIN {X 0,Y 414.738,Z 713.957,A -85,B 0,C 180,E1 16210.177,E2 16210.177} C_VEL
LIN {X 0,Y 427.331,Z 501.187,A -85,B 0,C 180,E1 16205.943,E2 16205.943} C_VEL
LIN {X 0,Y 428.713,Z 477.927,A -85,B 0,C 180,E1 16205.454,E2 16205.454} C_VEL
LIN {X 0,Y 421.417,Z 466.51,A -85,B 0,C 180,E1 16203.231,E2 16203.231} C_VEL
LIN {X 0,Y 415.8,Z 458.201,A -85,B 0,C 180,E1 16201.275,E2 16201.275} C_VEL
LIN {X 0,Y 412.269,Z 453.183,A -85,B 0,C 180,E1 16199.896,E2 16199.896} C_VEL
LIN {X 0,Y 409.746,Z 449.623,A -85,B 0,C 180,E1 16198.812,E2 16198.812} C_VEL
LIN {X 0,Y 406.657,Z 445.27,A -85,B 0,C 180,E1 16197.323,E2 16197.323} C_VEL
LIN {X 0,Y 403.389,Z 440.597,A -85,B 0,C 180,E1 16195.487,E2 16195.487} C_VEL
LIN {X 0,Y 399.99,Z 436.598,A -85,B 0,C 180,E1 16193.109,E2 16193.109} C_VEL
LIN {X 0,Y 399.085,Z 434.723,A -85,B 0,C 180,E1 16192.225,E2 16192.225} C_VEL
LIN {X 0,Y 395.983,Z 431.659,A -85,B 0,C 180,E1 16187.459,E2 16187.459} C_VEL
LIN {X 0,Y 395.92,Z 431.518,A -85,B 0,C 180,E1 16185.373,E2 16185.373} C_VEL
LIN {X 0,Y 398.569,Z 434.461,A -85,B 0,C 180,E1 16180.663,E2 16180.663} C_VEL
LIN {X 0,Y 399.401,Z 435.251,A -85,B 0,C 180,E1 16179.901,E2 16179.901} C_VEL
LIN {X 0,Y 401.7,Z 439.093,A -85,B 0,C 180,E1 16178.001,E2 16178.001} C_VEL
LIN {X 0,Y 403.5,Z 440.891,A -85,B 0,C 180,E1 16176.874,E2 16176.874} C_VEL
LIN {X 0,Y 406.731,Z 445.417,A -85,B 0,C 180,E1 16175.065,E2 16175.065} C_VEL
LIN {X 0,Y 410.603,Z 451.38,A -85,B 0,C 180,E1 16173.225,E2 16173.225} C_VEL
LIN {X 0,Y 415.388,Z 458.879,A -85,B 0,C 180,E1 16171.262,E2 16171.262} C_VEL
LIN {X 0,Y 422.163,Z 470.285,A -85,B 0,C 180,E1 16168.876,E2 16168.876} C_VEL
LIN {X 0,Y 428.746,Z 482.085,A -85,B 0,C 180,E1 16166.848,E2 16166.848} C_VEL
LIN {X 0,Y 417.461,Z 672.042,A -85,B 0,C 180,E1 16163.067,E2 16163.067} C_VEL
LIN {X 0,Y 413.737,Z 736.458,A -85,B 0,C 180,E1 16161.77,E2 16161.77} C_VEL
LIN {X 0,Y 411.108,Z 759.656,A -85,B 0,C 180,E1 16161.122,E2 16161.122} C_VEL
LIN {X 0,Y 407.83,Z 782.101,A -85,B 0,C 180,E1 16160.287,E2 16160.287} C_VEL
LIN {X 0,Y 404.194,Z 802.317,A -85,B 0,C 180,E1 16159.309,E2 16159.309} C_VEL
LIN {X 0,Y 399.907,Z 823.328,A -85,B 0,C 180,E1 16158.062,E2 16158.062} C_VEL
LIN {X 0,Y 395.133,Z 843.682,A -85,B 0,C 180,E1 16156.576,E2 16156.576} C_VEL
LIN {X 0,Y 389.845,Z 864.478,A -85,B 0,C 180,E1 16154.755,E2 16154.755} C_VEL
LIN {X 0,Y 384.572,Z 883.69,A -85,B 0,C 180,E1 16152.737,E2 16152.737} C_VEL
LIN {X 0,Y 379.227,Z 902.181,A -85,B 0,C 180,E1 16150.44,E2 16150.44} C_VEL
LIN {X 0,Y 374.12,Z 919.398,A -85,B 0,C 180,E1 16147.933,E2 16147.933} C_VEL
LIN {X 0,Y 369.255,Z 935.604,A -85,B 0,C 180,E1 16145.141,E2 16145.141} C_VEL
LIN {X 0,Y 364.85,Z 950.681,A -85,B 0,C 180,E1 16142.121,E2 16142.121} C_VEL
LIN {X 0,Y 361.123,Z 963.941,A -85,B 0,C 180,E1 16138.965,E2 16138.965} C_VEL
LIN {X 0,Y 357.782,Z 976.945,A -85,B 0,C 180,E1 16135.318,E2 16135.318} C_VEL
LIN {X 0,Y 355.519,Z 986.959,A -85,B 0,C 180,E1 16131.97,E2 16131.97} C_VEL
LIN {X 0,Y 353.777,Z 996.083,A -85,B 0,C 180,E1 16128.267,E2 16128.267} C_VEL
LIN {X 0,Y 352.782,Z 1002.899,A -85,B 0,C 180,E1 16124.882,E2 16124.882} C_VEL
LIN {X 0,Y 352.212,Z 1008.487,A -85,B 0,C 180,E1 16121.301,E2 16121.301} C_VEL
LIN {X 0,Y 352.017,Z 1012.128,A -85,B 0,C 180,E1 16118.169,E2 16118.169} C_VEL
LIN {X 0,Y 351.931,Z 1014.919,A -85,B 0,C 180,E1 16114.567,E2 16114.567} C_VEL
LIN {X 0,Y 351.935,Z 1016.028,A -85,B 0,C 180,E1 16111.307,E2 16111.307} C_VEL
LIN {X 0,Y 351.937,Z 1015.975,A -85,B 0,C 180,E1 16108.214,E2 16108.214} C_VEL
LIN {X 0,Y 351.935,Z 1014.472,A -85,B 0,C 180,E1 16104.626,E2 16104.626} C_VEL
LIN {X 0,Y 352.035,Z 1011.647,A -85,B 0,C 180,E1 16101.26,E2 16101.26} C_VEL
LIN {X 0,Y 352.363,Z 1007.039,A -85,B 0,C 180,E1 16097.552,E2 16097.552} C_VEL
LIN {X 0,Y 353.062,Z 1001.105,A -85,B 0,C 180,E1 16094.062,E2 16094.062} C_VEL
LIN {X 0,Y 354.423,Z 992.854,A -85,B 0,C 180,E1 16090.219,E2 16090.219} C_VEL
LIN {X 0,Y 356.247,Z 984.007,A -85,B 0,C 180,E1 16086.869,E2 16086.869} C_VEL
LIN {X 0,Y 359.069,Z 972.311,A -85,B 0,C 180,E1 16083.192,E2 16083.192} C_VEL
LIN {X 0,Y 362.467,Z 959.79,A -85,B 0,C 180,E1 16079.872,E2 16079.872} C_VEL
LIN {X 0,Y 366.484,Z 945.737,A -85,B 0,C 180,E1 16076.751,E2 16076.751} C_VEL
LIN {X 0,Y 371.115,Z 930.151,A -85,B 0,C 180,E1 16073.786,E2 16073.786} C_VEL
LIN {X 0,Y 375.892,Z 914.113,A -85,B 0,C 180,E1 16071.202,E2 16071.202} C_VEL
LIN {X 0,Y 381.315,Z 895.495,A -85,B 0,C 180,E1 16068.649,E2 16068.649} C_VEL
LIN {X 0,Y 386.476,Z 877.172,A -85,B 0,C 180,E1 16066.523,E2 16066.523} C_VEL
LIN {X 0,Y 391.671,Z 857.268,A -85,B 0,C 180,E1 16064.592,E2 16064.592} C_VEL
LIN {X 0,Y 396.63,Z 836.894,A -85,B 0,C 180,E1 16062.928,E2 16062.928} C_VEL
LIN {X 0,Y 401.053,Z 816.1,A -85,B 0,C 180,E1 16061.54,E2 16061.54} C_VEL
LIN {X 0,Y 405.109,Z 794.631,A -85,B 0,C 180,E1 16060.366,E2 16060.366} C_VEL
LIN {X 0,Y 408.51,Z 772.75,A -85,B 0,C 180,E1 16059.429,E2 16059.429} C_VEL
LIN {X 0,Y 411.546,Z 748.055,A -85,B 0,C 180,E1 16058.644,E2 16058.644} C_VEL
LIN {X 0,Y 413.392,Z 724.96,A -85,B 0,C 180,E1 16058.112,E2 16058.112} C_VEL
LIN {X 0,Y 424.084,Z 516.138,A -85,B 0,C 180,E1 16054.071,E2 16054.071} C_VEL
LIN {X 0,Y 425.811,Z 481.595,A -85,B 0,C 180,E1 16053.37,E2 16053.37} C_VEL
LIN {X 0,Y 414.037,Z 463.084,A -85,B 0,C 180,E1 16050.392,E2 16050.392} C_VEL
LIN {X 0,Y 403.324,Z 447.497,A -85,B 0,C 180,E1 16047.378,E2 16047.378} C_VEL
LIN {X 0,Y 396.592,Z 438.287,A -85,B 0,C 180,E1 16045.298,E2 16045.298} C_VEL
LIN {X 0,Y 390.239,Z 429.724,A -85,B 0,C 180,E1 16043.159,E2 16043.159} C_VEL
LIN {X 0,Y 386.036,Z 424.513,A -85,B 0,C 180,E1 16041.659,E2 16041.659} C_VEL
LIN {X 0,Y 382.379,Z 420.074,A -85,B 0,C 180,E1 16040.271,E2 16040.271} C_VEL
LIN {X 0,Y 380.75,Z 418.37,A -85,B 0,C 180,E1 16039.641,E2 16039.641} C_VEL
LIN {X 0,Y 377.39,Z 414.287,A -85,B 0,C 180,E1 16038.257,E2 16038.257} C_VEL
LIN {X 0,Y 376.315,Z 412.91,A -85,B 0,C 180,E1 16037.791,E2 16037.791} C_VEL
LIN {X 0,Y 372.939,Z 409.539,A -85,B 0,C 180,E1 16036.31,E2 16036.31} C_VEL
LIN {X 0,Y 371.211,Z 406.805,A -85,B 0,C 180,E1 16035.465,E2 16035.465} C_VEL
LIN {X 0,Y 367.811,Z 404.054,A -85,B 0,C 180,E1 16033.84,E2 16033.84} C_VEL
LIN {X 0,Y 365.663,Z 400.423,A -85,B 0,C 180,E1 16032.635,E2 16032.635} C_VEL
LIN {X 0,Y 362.164,Z 397.986,A -85,B 0,C 180,E1 16030.739,E2 16030.739} C_VEL
LIN {X 0,Y 360.255,Z 394.908,A -85,B 0,C 180,E1 16029.505,E2 16029.505} C_VEL
LIN {X 0,Y 359.438,Z 393.7,A -85,B 0,C 180,E1 16028.961,E2 16028.961} C_VEL
LIN {X 0,Y 355.868,Z 391.405,A -85,B 0,C 180,E1 16026.614,E2 16026.614} C_VEL
LIN {X 0,Y 354.166,Z 388.419,A -85,B 0,C 180,E1 16025.183,E2 16025.183} C_VEL
LIN {X 0,Y 353.823,Z 387.085,A -85,B 0,C 180,E1 16024.05,E2 16024.05} C_VEL
LIN {X 0,Y 353.809,Z 386.97,A -85,B 0,C 180,E1 16019.999,E2 16019.999} C_VEL
LIN {X 0,Y 353.813,Z 386.961,A -85,B 0,C 180,E1 16015.786,E2 16015.786} C_VEL
LIN {X 0,Y 353.815,Z 386.959,A -85,B 0,C 180,E1 16011.713,E2 16011.713} C_VEL
LIN {X 0,Y 353.819,Z 386.965,A -85,B 0,C 180,E1 16007.597,E2 16007.597} C_VEL
LIN {X 0,Y 353.825,Z 386.976,A -85,B 0,C 180,E1 16003.416,E2 16003.416} C_VEL
LIN {X 0,Y 353.828,Z 386.964,A -85,B 0,C 180,E1 15999.265,E2 15999.265} C_VEL
LIN {X 0,Y 353.831,Z 386.957,A -85,B 0,C 180,E1 15995.099,E2 15995.099} C_VEL
LIN {X 0,Y 353.835,Z 386.959,A -85,B 0,C 180,E1 15990.919,E2 15990.919} C_VEL
LIN {X 0,Y 353.859,Z 387.158,A -85,B 0,C 180,E1 15987.043,E2 15987.043} C_VEL
LIN {X 0,Y 354.163,Z 388.34,A -85,B 0,C 180,E1 15986.087,E2 15986.087} C_VEL
LIN {X 0,Y 355.751,Z 391.23,A -85,B 0,C 180,E1 15984.719,E2 15984.719} C_VEL
LIN {X 0,Y 358.944,Z 393.478,A -85,B 0,C 180,E1 15982.608,E2 15982.608} C_VEL
LIN {X 0,Y 360.14,Z 394.531,A -85,B 0,C 180,E1 15981.849,E2 15981.849} C_VEL
LIN {X 0,Y 361.95,Z 397.734,A -85,B 0,C 180,E1 15980.657,E2 15980.657} C_VEL
LIN {X 0,Y 365.332,Z 400.25,A -85,B 0,C 180,E1 15978.809,E2 15978.809} C_VEL
LIN {X 0,Y 365.989,Z 400.958,A -85,B 0,C 180,E1 15978.455,E2 15978.455} C_VEL
LIN {X 0,Y 368.208,Z 404.476,A -85,B 0,C 180,E1 15977.244,E2 15977.244} C_VEL
LIN {X 0,Y 371.55,Z 407.198,A -85,B 0,C 180,E1 15975.665,E2 15975.665} C_VEL
LIN {X 0,Y 374.332,Z 411.207,A -85,B 0,C 180,E1 15974.347,E2 15974.347} C_VEL
LIN {X 0,Y 377.091,Z 413.73,A -85,B 0,C 180,E1 15973.183,E2 15973.183} C_VEL
LIN {X 0,Y 380.146,Z 417.785,A -85,B 0,C 180,E1 15971.896,E2 15971.896} C_VEL
LIN {X 0,Y 382.267,Z 419.881,A -85,B 0,C 180,E1 15971.083,E2 15971.083} C_VEL
LIN {X 0,Y 385.922,Z 424.391,A -85,B 0,C 180,E1 15969.692,E2 15969.692} C_VEL
LIN {X 0,Y 387.794,Z 426.707,A -85,B 0,C 180,E1 15969.014,E2 15969.014} C_VEL
LIN {X 0,Y 392.443,Z 432.281,A -85,B 0,C 180,E1 15967.413,E2 15967.413} C_VEL
LIN {X 0,Y 397.115,Z 438.148,A -85,B 0,C 180,E1 15965.899,E2 15965.899} C_VEL
LIN {X 0,Y 405.178,Z 448.461,A -85,B 0,C 180,E1 15963.479,E2 15963.479} C_VEL
LIN {X 0,Y 415.812,Z 462.893,A -85,B 0,C 180,E1 15960.587,E2 15960.587} C_VEL
LIN {X 0,Y 425.64,Z 477.128,A -85,B 0,C 180,E1 15958.16,E2 15958.16} C_VEL
LIN {X 0,Y 414.803,Z 685.184,A -85,B 0,C 180,E1 15954.138,E2 15954.138} C_VEL
LIN {X 0,Y 412.715,Z 720.124,A -85,B 0,C 180,E1 15953.419,E2 15953.419} C_VEL
LIN {X 0,Y 410.405,Z 742.088,A -85,B 0,C 180,E1 15952.776,E2 15952.776} C_VEL
LIN {X 0,Y 407.168,Z 765.522,A -85,B 0,C 180,E1 15951.843,E2 15951.843} C_VEL
LIN {X 0,Y 403.714,Z 785.778,A -85,B 0,C 180,E1 15950.812,E2 15950.812} C_VEL
LIN {X 0,Y 399.355,Z 807.435,A -85,B 0,C 180,E1 15949.445,E2 15949.445} C_VEL
LIN {X 0,Y 394.989,Z 826.608,A -85,B 0,C 180,E1 15947.983,E2 15947.983} C_VEL
LIN {X 0,Y 389.883,Z 846.604,A -85,B 0,C 180,E1 15946.15,E2 15946.15} C_VEL
LIN {X 0,Y 388.809,Z 850.617,A -85,B 0,C 180,E1 15945.746,E2 15945.746} C_VEL
LIN {X 0,Y 386.375,Z 856.952,A -85,B 0,C 180,E1 15945.186,E2 15945.186} C_VEL
LIN {X 0,Y 377.244,Z 872.828,A -85,B 0,C 180,E1 15943.936,E2 15943.936} C_VEL
LIN {X 0,Y 374.628,Z 878.639,A -85,B 0,C 180,E1 15943.263,E2 15943.263} C_VEL
LIN {X 0,Y 369.53,Z 894.639,A -85,B 0,C 180,E1 15940.913,E2 15940.913} C_VEL
LIN {X 0,Y 364.162,Z 911.234,A -85,B 0,C 180,E1 15938.044,E2 15938.044} C_VEL
LIN {X 0,Y 359.675,Z 924.92,A -85,B 0,C 180,E1 15935.258,E2 15935.258} C_VEL
LIN {X 0,Y 355.254,Z 938.744,A -85,B 0,C 180,E1 15931.93,E2 15931.93} C_VEL
LIN {X 0,Y 351.665,Z 950.674,A -85,B 0,C 180,E1 15928.529,E2 15928.529} C_VEL
LIN {X 0,Y 348.841,Z 960.697,A -85,B 0,C 180,E1 15925.062,E2 15925.062} C_VEL
LIN {X 0,Y 346.773,Z 969.385,A -85,B 0,C 180,E1 15921.49,E2 15921.49} C_VEL
LIN {X 0,Y 345.346,Z 976.51,A -85,B 0,C 180,E1 15917.794,E2 15917.794} C_VEL
LIN {X 0,Y 344.485,Z 982.297,A -85,B 0,C 180,E1 15913.99,E2 15913.99} C_VEL
LIN {X 0,Y 344.111,Z 985.966,A -85,B 0,C 180,E1 15910.651,E2 15910.651} C_VEL
LIN {X 0,Y 343.982,Z 988.561,A -85,B 0,C 180,E1 15907.253,E2 15907.253} C_VEL
LIN {X 0,Y 343.93,Z 989.901,A -85,B 0,C 180,E1 15903.562,E2 15903.562} C_VEL
LIN {X 0,Y 343.933,Z 989.925,A -85,B 0,C 180,E1 15900.378,E2 15900.378} C_VEL
LIN {X 0,Y 343.976,Z 988.752,A -85,B 0,C 180,E1 15896.841,E2 15896.841} C_VEL
LIN {X 0,Y 344.114,Z 986.139,A -85,B 0,C 180,E1 15893.318,E2 15893.318} C_VEL
LIN {X 0,Y 344.56,Z 982.171,A -85,B 0,C 180,E1 15889.671,E2 15889.671} C_VEL
LIN {X 0,Y 345.406,Z 976.53,A -85,B 0,C 180,E1 15885.989,E2 15885.989} C_VEL
LIN {X 0,Y 346.857,Z 969.518,A -85,B 0,C 180,E1 15882.328,E2 15882.328} C_VEL
LIN {X 0,Y 348.945,Z 960.969,A -85,B 0,C 180,E1 15878.791,E2 15878.791} C_VEL
LIN {X 0,Y 351.902,Z 950.704,A -85,B 0,C 180,E1 15875.225,E2 15875.225} C_VEL
LIN {X 0,Y 355.451,Z 939.238,A -85,B 0,C 180,E1 15871.927,E2 15871.927} C_VEL
LIN {X 0,Y 360.038,Z 925.273,A -85,B 0,C 180,E1 15868.533,E2 15868.533} C_VEL
LIN {X 0,Y 364.772,Z 911.279,A -85,B 0,C 180,E1 15865.664,E2 15865.664} C_VEL
LIN {X 0,Y 370.094,Z 895.268,A -85,B 0,C 180,E1 15862.883,E2 15862.883} C_VEL
LIN {X 0,Y 375.608,Z 878.551,A -85,B 0,C 180,E1 15860.41,E2 15860.41} C_VEL
LIN {X 0,Y 381.115,Z 860.677,A -85,B 0,C 180,E1 15858.192,E2 15858.192} C_VEL
LIN {X 0,Y 386.565,Z 842.029,A -85,B 0,C 180,E1 15856.222,E2 15856.222} C_VEL
LIN {X 0,Y 391.766,Z 822.277,A -85,B 0,C 180,E1 15854.485,E2 15854.485} C_VEL
LIN {X 0,Y 397.111,Z 799.564,A -85,B 0,C 180,E1 15852.842,E2 15852.842} C_VEL
LIN {X 0,Y 401.438,Z 778.411,A -85,B 0,C 180,E1 15851.603,E2 15851.603} C_VEL
LIN {X 0,Y 405.088,Z 756.512,A -85,B 0,C 180,E1 15850.592,E2 15850.592} C_VEL
LIN {X 0,Y 408.143,Z 733.955,A -85,B 0,C 180,E1 15849.788,E2 15849.788} C_VEL
LIN {X 0,Y 410.218,Z 711.289,A -85,B 0,C 180,E1 15849.216,E2 15849.216} C_VEL
LIN {X 0,Y 423.169,Z 502.89,A -85,B 0,C 180,E1 15845.041,E2 15845.041} C_VEL
LIN {X 0,Y 424.482,Z 482.439,A -85,B 0,C 180,E1 15844.616,E2 15844.616} C_VEL
LIN {X 0,Y 417.362,Z 471.054,A -85,B 0,C 180,E1 15842.297,E2 15842.297} C_VEL
LIN {X 0,Y 411.216,Z 461.885,A -85,B 0,C 180,E1 15839.966,E2 15839.966} C_VEL
LIN {X 0,Y 407.764,Z 456.949,A -85,B 0,C 180,E1 15838.455,E2 15838.455} C_VEL
LIN {X 0,Y 404.764,Z 452.651,A -85,B 0,C 180,E1 15836.956,E2 15836.956} C_VEL
LIN {X 0,Y 401.475,Z 447.911,A -85,B 0,C 180,E1 15835,E2 15835} C_VEL
LIN {X 0,Y 398.503,Z 444.146,A -85,B 0,C 180,E1 15832.794,E2 15832.794} C_VEL
LIN {X 0,Y 397.788,Z 442.558,A -85,B 0,C 180,E1 15832.043,E2 15832.043} C_VEL
LIN {X 0,Y 394.839,Z 439.481,A -85,B 0,C 180,E1 15827.124,E2 15827.124} C_VEL
LIN {X 0,Y 394.866,Z 439.519,A -85,B 0,C 180,E1 15825.183,E2 15825.183} C_VEL
LIN {X 0,Y 397.898,Z 442.642,A -85,B 0,C 180,E1 15820.285,E2 15820.285} C_VEL
LIN {X 0,Y 400.161,Z 446.692,A -85,B 0,C 180,E1 15818.297,E2 15818.297} C_VEL
LIN {X 0,Y 401.941,Z 448.607,A -85,B 0,C 180,E1 15817.128,E2 15817.128} C_VEL
LIN {X 0,Y 406.018,Z 454.561,A -85,B 0,C 180,E1 15814.824,E2 15814.824} C_VEL
LIN {X 0,Y 410.843,Z 462.37,A -85,B 0,C 180,E1 15812.577,E2 15812.577} C_VEL
LIN {X 0,Y 415.705,Z 470.547,A -85,B 0,C 180,E1 15810.656,E2 15810.656} C_VEL
LIN {X 0,Y 422.342,Z 482.234,A -85,B 0,C 180,E1 15808.374,E2 15808.374} C_VEL
LIN {X 0,Y 424.459,Z 486.512,A -85,B 0,C 180,E1 15807.695,E2 15807.695} C_VEL
LIN {X 0,Y 412.595,Z 676.753,A -85,B 0,C 180,E1 15803.882,E2 15803.882} C_VEL
LIN {X 0,Y 408.902,Z 736.613,A -85,B 0,C 180,E1 15802.66,E2 15802.66} C_VEL
LIN {X 0,Y 406.197,Z 759.583,A -85,B 0,C 180,E1 15802.015,E2 15802.015} C_VEL
LIN {X 0,Y 402.737,Z 782.209,A -85,B 0,C 180,E1 15801.167,E2 15801.167} C_VEL
LIN {X 0,Y 398.968,Z 802.294,A -85,B 0,C 180,E1 15800.19,E2 15800.19} C_VEL
LIN {X 0,Y 394.267,Z 824.221,A -85,B 0,C 180,E1 15798.872,E2 15798.872} C_VEL
LIN {X 0,Y 389.553,Z 843.502,A -85,B 0,C 180,E1 15797.45,E2 15797.45} C_VEL
LIN {X 0,Y 383.816,Z 864.973,A -85,B 0,C 180,E1 15795.548,E2 15795.548} C_VEL
LIN {X 0,Y 378.515,Z 883.416,A -85,B 0,C 180,E1 15793.59,E2 15793.59} C_VEL
LIN {X 0,Y 372.722,Z 902.501,A -85,B 0,C 180,E1 15791.183,E2 15791.183} C_VEL
LIN {X 0,Y 367.363,Z 919.71,A -85,B 0,C 180,E1 15788.637,E2 15788.637} C_VEL
LIN {X 0,Y 362.141,Z 936.155,A -85,B 0,C 180,E1 15785.737,E2 15785.737} C_VEL
LIN {X 0,Y 357.531,Z 951.054,A -85,B 0,C 180,E1 15782.67,E2 15782.67} C_VEL
LIN {X 0,Y 353.597,Z 964.322,A -85,B 0,C 180,E1 15779.435,E2 15779.435} C_VEL
LIN {X 0,Y 350.097,Z 977.131,A -85,B 0,C 180,E1 15775.733,E2 15775.733} C_VEL
LIN {X 0,Y 347.611,Z 987.566,A -85,B 0,C 180,E1 15772.14,E2 15772.14} C_VEL
LIN {X 0,Y 345.872,Z 996.113,A -85,B 0,C 180,E1 15768.526,E2 15768.526} C_VEL
LIN {X 0,Y 344.797,Z 1003.07,A -85,B 0,C 180,E1 15764.961,E2 15764.961} C_VEL
LIN {X 0,Y 344.22,Z 1008.383,A -85,B 0,C 180,E1 15761.397,E2 15761.397} C_VEL
LIN {X 0,Y 344.006,Z 1012.148,A -85,B 0,C 180,E1 15758.024,E2 15758.024} C_VEL
LIN {X 0,Y 343.937,Z 1014.758,A -85,B 0,C 180,E1 15754.34,E2 15754.34} C_VEL
LIN {X 0,Y 343.936,Z 1015.751,A -85,B 0,C 180,E1 15751.171,E2 15751.171} C_VEL
LIN {X 0,Y 343.943,Z 1015.63,A -85,B 0,C 180,E1 15747.839,E2 15747.839} C_VEL
LIN {X 0,Y 343.943,Z 1013.939,A -85,B 0,C 180,E1 15744.166,E2 15744.166} C_VEL
LIN {X 0,Y 344.056,Z 1011.103,A -85,B 0,C 180,E1 15740.808,E2 15740.808} C_VEL
LIN {X 0,Y 344.455,Z 1006.207,A -85,B 0,C 180,E1 15736.92,E2 15736.92} C_VEL
LIN {X 0,Y 345.227,Z 1000.384,A -85,B 0,C 180,E1 15733.464,E2 15733.464} C_VEL
LIN {X 0,Y 346.709,Z 992.113,A -85,B 0,C 180,E1 15729.583,E2 15729.583} C_VEL
LIN {X 0,Y 348.714,Z 983.184,A -85,B 0,C 180,E1 15726.156,E2 15726.156} C_VEL
LIN {X 0,Y 351.676,Z 971.703,A -85,B 0,C 180,E1 15722.504,E2 15722.504} C_VEL
LIN {X 0,Y 355.305,Z 959.152,A -85,B 0,C 180,E1 15719.125,E2 15719.125} C_VEL
LIN {X 0,Y 359.548,Z 945.083,A -85,B 0,C 180,E1 15715.964,E2 15715.964} C_VEL
LIN {X 0,Y 364.567,Z 929.071,A -85,B 0,C 180,E1 15712.896,E2 15712.896} C_VEL
LIN {X 0,Y 369.361,Z 913.756,A -85,B 0,C 180,E1 15710.403,E2 15710.403} C_VEL
LIN {X 0,Y 375.075,Z 894.968,A -85,B 0,C 180,E1 15707.804,E2 15707.804} C_VEL
LIN {X 0,Y 380.48,Z 876.601,A -85,B 0,C 180,E1 15705.66,E2 15705.66} C_VEL
LIN {X 0,Y 385.605,Z 857.736,A -85,B 0,C 180,E1 15703.813,E2 15703.813} C_VEL
LIN {X 0,Y 390.589,Z 838.113,A -85,B 0,C 180,E1 15702.185,E2 15702.185} C_VEL
LIN {X 0,Y 395.204,Z 817.392,A -85,B 0,C 180,E1 15700.777,E2 15700.777} C_VEL
LIN {X 0,Y 399.477,Z 795.864,A -85,B 0,C 180,E1 15699.575,E2 15699.575} C_VEL
LIN {X 0,Y 403.122,Z 773.227,A -85,B 0,C 180,E1 15698.595,E2 15698.595} C_VEL
LIN {X 0,Y 406.184,Z 749.7,A -85,B 0,C 180,E1 15697.83,E2 15697.83} C_VEL
LIN {X 0,Y 408.112,Z 727.217,A -85,B 0,C 180,E1 15697.299,E2 15697.299} C_VEL
LIN {X 0,Y 419.377,Z 516.958,A -85,B 0,C 180,E1 15693.199,E2 15693.199} C_VEL
LIN {X 0,Y 421.065,Z 485.787,A -85,B 0,C 180,E1 15692.577,E2 15692.577} C_VEL
LIN {X 0,Y 410.318,Z 468.811,A -85,B 0,C 180,E1 15689.768,E2 15689.768} C_VEL
LIN {X 0,Y 400.329,Z 454.043,A -85,B 0,C 180,E1 15686.876,E2 15686.876} C_VEL
LIN {X 0,Y 393.486,Z 444.596,A -85,B 0,C 180,E1 15684.708,E2 15684.708} C_VEL
LIN {X 0,Y 387.615,Z 436.631,A -85,B 0,C 180,E1 15682.683,E2 15682.683} C_VEL
LIN {X 0,Y 383.665,Z 431.669,A -85,B 0,C 180,E1 15681.237,E2 15681.237} C_VEL
LIN {X 0,Y 379.891,Z 426.902,A -85,B 0,C 180,E1 15679.767,E2 15679.767} C_VEL
LIN {X 0,Y 375.713,Z 422.276,A -85,B 0,C 180,E1 15678.061,E2 15678.061} C_VEL
LIN {X 0,Y 374.422,Z 420.45,A -85,B 0,C 180,E1 15677.482,E2 15677.482} C_VEL
LIN {X 0,Y 370.834,Z 416.743,A -85,B 0,C 180,E1 15675.882,E2 15675.882} C_VEL
LIN {X 0,Y 369.198,Z 414.297,A -85,B 0,C 180,E1 15675.069,E2 15675.069} C_VEL
LIN {X 0,Y 365.871,Z 411.372,A -85,B 0,C 180,E1 15673.431,E2 15673.431} C_VEL
LIN {X 0,Y 363.72,Z 408.002,A -85,B 0,C 180,E1 15672.22,E2 15672.22} C_VEL
LIN {X 0,Y 360.192,Z 405.198,A -85,B 0,C 180,E1 15670.233,E2 15670.233} C_VEL
LIN {X 0,Y 358.272,Z 401.796,A -85,B 0,C 180,E1 15668.937,E2 15668.937} C_VEL
LIN {X 0,Y 354.132,Z 398.8,A -85,B 0,C 180,E1 15666.158,E2 15666.158} C_VEL
LIN {X 0,Y 351.915,Z 395.028,A -85,B 0,C 180,E1 15664.236,E2 15664.236} C_VEL
LIN {X 0,Y 347.499,Z 391.893,A -85,B 0,C 180,E1 15660.164,E2 15660.164} C_VEL
LIN {X 0,Y 346.015,Z 388.755,A -85,B 0,C 180,E1 15657.846,E2 15657.846} C_VEL
LIN {X 0,Y 345.878,Z 387.994,A -85,B 0,C 180,E1 15656.021,E2 15656.021} C_VEL
LIN {X 0,Y 345.877,Z 387.948,A -85,B 0,C 180,E1 15651.689,E2 15651.689} C_VEL
LIN {X 0,Y 345.884,Z 387.955,A -85,B 0,C 180,E1 15647.478,E2 15647.478} C_VEL
LIN {X 0,Y 345.888,Z 387.965,A -85,B 0,C 180,E1 15643.37,E2 15643.37} C_VEL
LIN {X 0,Y 345.891,Z 387.951,A -85,B 0,C 180,E1 15639.172,E2 15639.172} C_VEL
LIN {X 0,Y 345.9,Z 387.998,A -85,B 0,C 180,E1 15635.037,E2 15635.037} C_VEL
LIN {X 0,Y 346.114,Z 389.064,A -85,B 0,C 180,E1 15633.028,E2 15633.028} C_VEL
LIN {X 0,Y 348.117,Z 392.524,A -85,B 0,C 180,E1 15630.394,E2 15630.394} C_VEL
LIN {X 0,Y 352.314,Z 395.378,A -85,B 0,C 180,E1 15626.691,E2 15626.691} C_VEL
LIN {X 0,Y 354.335,Z 398.982,A -85,B 0,C 180,E1 15624.943,E2 15624.943} C_VEL
LIN {X 0,Y 357.485,Z 401.267,A -85,B 0,C 180,E1 15622.832,E2 15622.832} C_VEL
LIN {X 0,Y 358.404,Z 402.018,A -85,B 0,C 180,E1 15622.24,E2 15622.24} C_VEL
LIN {X 0,Y 360.45,Z 405.497,A -85,B 0,C 180,E1 15620.87,E2 15620.87} C_VEL
LIN {X 0,Y 364.142,Z 408.482,A -85,B 0,C 180,E1 15618.829,E2 15618.829} C_VEL
LIN {X 0,Y 366.653,Z 412.252,A -85,B 0,C 180,E1 15617.445,E2 15617.445} C_VEL
LIN {X 0,Y 369.723,Z 414.898,A -85,B 0,C 180,E1 15615.971,E2 15615.971} C_VEL
LIN {X 0,Y 372.835,Z 419.095,A -85,B 0,C 180,E1 15614.491,E2 15614.491} C_VEL
LIN {X 0,Y 375.094,Z 421.237,A -85,B 0,C 180,E1 15613.526,E2 15613.526} C_VEL
LIN {X 0,Y 378.513,Z 425.582,A -85,B 0,C 180,E1 15612.074,E2 15612.074} C_VEL
LIN {X 0,Y 380.322,Z 427.587,A -85,B 0,C 180,E1 15611.359,E2 15611.359} C_VEL
LIN {X 0,Y 384.26,Z 432.191,A -85,B 0,C 180,E1 15609.86,E2 15609.86} C_VEL
LIN {X 0,Y 388.947,Z 437.933,A -85,B 0,C 180,E1 15608.187,E2 15608.187} C_VEL
LIN {X 0,Y 397.919,Z 449.451,A -85,B 0,C 180,E1 15605.25,E2 15605.25} C_VEL
LIN {X 0,Y 406.615,Z 461.097,A -85,B 0,C 180,E1 15602.691,E2 15602.691} C_VEL
LIN {X 0,Y 416.064,Z 474.369,A -85,B 0,C 180,E1 15600.163,E2 15600.163} C_VEL
LIN {X 0,Y 420.81,Z 481.624,A -85,B 0,C 180,E1 15598.966,E2 15598.966} C_VEL
LIN {X 0,Y 409.505,Z 690.19,A -85,B 0,C 180,E1 15594.908,E2 15594.908} C_VEL
LIN {X 0,Y 407.416,Z 722.058,A -85,B 0,C 180,E1 15594.233,E2 15594.233} C_VEL
LIN {X 0,Y 405.01,Z 743.924,A -85,B 0,C 180,E1 15593.578,E2 15593.578} C_VEL
LIN {X 0,Y 401.687,Z 766.761,A -85,B 0,C 180,E1 15592.65,E2 15592.65} C_VEL
LIN {X 0,Y 398.038,Z 787.403,A -85,B 0,C 180,E1 15591.587,E2 15591.587} C_VEL
LIN {X 0,Y 393.52,Z 808.833,A -85,B 0,C 180,E1 15590.21,E2 15590.21} C_VEL
LIN {X 0,Y 388.807,Z 828.732,A -85,B 0,C 180,E1 15588.667,E2 15588.667} C_VEL
LIN {X 0,Y 383.506,Z 848.424,A -85,B 0,C 180,E1 15586.816,E2 15586.816} C_VEL
LIN {X 0,Y 378.033,Z 867.422,A -85,B 0,C 180,E1 15584.704,E2 15584.704} C_VEL
LIN {X 0,Y 374.628,Z 878.639,A -85,B 0,C 180,E1 15583.263,E2 15583.263} C_VEL
LIN {X 0,Y 372.001,Z 884.42,A -85,B 0,C 180,E1 15582.56,E2 15582.56} C_VEL
LIN {X 0,Y 362.543,Z 898.944,A -85,B 0,C 180,E1 15580.955,E2 15580.955} C_VEL
LIN {X 0,Y 359.956,Z 904.101,A -85,B 0,C 180,E1 15580.156,E2 15580.156} C_VEL
LIN {X 0,Y 354.812,Z 919.193,A -85,B 0,C 180,E1 15577.28,E2 15577.28} C_VEL
LIN {X 0,Y 350.229,Z 932.525,A -85,B 0,C 180,E1 15574.252,E2 15574.252} C_VEL
LIN {X 0,Y 345.989,Z 945.436,A -85,B 0,C 180,E1 15570.799,E2 15570.799} C_VEL
LIN {X 0,Y 342.756,Z 955.807,A -85,B 0,C 180,E1 15567.487,E2 15567.487} C_VEL
LIN {X 0,Y 339.936,Z 965.948,A -85,B 0,C 180,E1 15563.578,E2 15563.578} C_VEL
LIN {X 0,Y 338.136,Z 973.641,A -85,B 0,C 180,E1 15559.948,E2 15559.948} C_VEL
LIN {X 0,Y 336.902,Z 980.128,A -85,B 0,C 180,E1 15556.044,E2 15556.044} C_VEL
LIN {X 0,Y 336.3,Z 984.845,A -85,B 0,C 180,E1 15552.342,E2 15552.342} C_VEL
LIN {X 0,Y 336.028,Z 988.106,A -85,B 0,C 180,E1 15548.527,E2 15548.527} C_VEL
LIN {X 0,Y 335.965,Z 989.806,A -85,B 0,C 180,E1 15545.184,E2 15545.184} C_VEL
LIN {X 0,Y 335.953,Z 990.352,A -85,B 0,C 180,E1 15541.364,E2 15541.364} C_VEL
LIN {X 0,Y 335.964,Z 989.583,A -85,B 0,C 180,E1 15538.007,E2 15538.007} C_VEL
LIN {X 0,Y 336.089,Z 987.517,A -85,B 0,C 180,E1 15534.31,E2 15534.31} C_VEL
LIN {X 0,Y 336.439,Z 983.781,A -85,B 0,C 180,E1 15530.502,E2 15530.502} C_VEL
LIN {X 0,Y 337.23,Z 978.804,A -85,B 0,C 180,E1 15526.768,E2 15526.768} C_VEL
LIN {X 0,Y 338.622,Z 971.922,A -85,B 0,C 180,E1 15522.917,E2 15522.917} C_VEL
LIN {X 0,Y 340.871,Z 963.186,A -85,B 0,C 180,E1 15518.98,E2 15518.98} C_VEL
LIN {X 0,Y 343.599,Z 953.975,A -85,B 0,C 180,E1 15515.592,E2 15515.592} C_VEL
LIN {X 0,Y 347.494,Z 942.012,A -85,B 0,C 180,E1 15511.911,E2 15511.911} C_VEL
LIN {X 0,Y 351.791,Z 929.612,A -85,B 0,C 180,E1 15508.708,E2 15508.708} C_VEL
LIN {X 0,Y 356.925,Z 915.071,A -85,B 0,C 180,E1 15505.557,E2 15505.557} C_VEL
LIN {X 0,Y 362.397,Z 899.715,A -85,B 0,C 180,E1 15502.723,E2 15502.723} C_VEL
LIN {X 0,Y 368.009,Z 883.318,A -85,B 0,C 180,E1 15500.186,E2 15500.186} C_VEL
LIN {X 0,Y 374.198,Z 864.601,A -85,B 0,C 180,E1 15497.735,E2 15497.735} C_VEL
LIN {X 0,Y 379.555,Z 847.247,A -85,B 0,C 180,E1 15495.823,E2 15495.823} C_VEL
LIN {X 0,Y 385.479,Z 826.236,A -85,B 0,C 180,E1 15493.883,E2 15493.883} C_VEL
LIN {X 0,Y 390.608,Z 806.083,A -85,B 0,C 180,E1 15492.342,E2 15492.342} C_VEL
LIN {X 0,Y 395.25,Z 784.793,A -85,B 0,C 180,E1 15491.021,E2 15491.021} C_VEL
LIN {X 0,Y 399.402,Z 762.556,A -85,B 0,C 180,E1 15489.911,E2 15489.911} C_VEL
LIN {X 0,Y 402.646,Z 740.318,A -85,B 0,C 180,E1 15489.063,E2 15489.063} C_VEL
LIN {X 0,Y 405.346,Z 715.303,A -85,B 0,C 180,E1 15488.377,E2 15488.377} C_VEL
LIN {X 0,Y 419.281,Z 502.947,A -85,B 0,C 180,E1 15484.086,E2 15484.086} C_VEL
LIN {X 0,Y 420.361,Z 486.963,A -85,B 0,C 180,E1 15483.751,E2 15483.751} C_VEL
LIN {X 0,Y 413.926,Z 476.588,A -85,B 0,C 180,E1 15481.523,E2 15481.523} C_VEL
LIN {X 0,Y 408.563,Z 468.401,A -85,B 0,C 180,E1 15479.37,E2 15479.37} C_VEL
LIN {X 0,Y 405.645,Z 464.077,A -85,B 0,C 180,E1 15478.023,E2 15478.023} C_VEL
LIN {X 0,Y 402.905,Z 460.029,A -85,B 0,C 180,E1 15476.586,E2 15476.586} C_VEL
LIN {X 0,Y 399.869,Z 455.512,A -85,B 0,C 180,E1 15474.692,E2 15474.692} C_VEL
LIN {X 0,Y 396.984,Z 451.541,A -85,B 0,C 180,E1 15472.402,E2 15472.402} C_VEL
LIN {X 0,Y 396.359,Z 450.319,A -85,B 0,C 180,E1 15471.733,E2 15471.733} C_VEL
LIN {X 0,Y 393.755,Z 447.404,A -85,B 0,C 180,E1 15467.088,E2 15467.088} C_VEL
LIN {X 0,Y 393.791,Z 447.47,A -85,B 0,C 180,E1 15465.141,E2 15465.141} C_VEL
LIN {X 0,Y 396.573,Z 450.498,A -85,B 0,C 180,E1 15460.485,E2 15460.485} C_VEL
LIN {X 0,Y 398.924,Z 454.626,A -85,B 0,C 180,E1 15458.381,E2 15458.381} C_VEL
LIN {X 0,Y 400.395,Z 456.309,A -85,B 0,C 180,E1 15457.384,E2 15457.384} C_VEL
LIN {X 0,Y 404.286,Z 462.174,A -85,B 0,C 180,E1 15455.1,E2 15455.1} C_VEL
LIN {X 0,Y 408.919,Z 469.95,A -85,B 0,C 180,E1 15452.87,E2 15452.87} C_VEL
LIN {X 0,Y 414.54,Z 479.694,A -85,B 0,C 180,E1 15450.605,E2 15450.605} C_VEL
LIN {X 0,Y 420.318,Z 490.605,A -85,B 0,C 180,E1 15448.569,E2 15448.569} C_VEL
LIN {X 0,Y 407.854,Z 680.88,A -85,B 0,C 180,E1 15444.729,E2 15444.729} C_VEL
LIN {X 0,Y 404.268,Z 736.228,A -85,B 0,C 180,E1 15443.589,E2 15443.589} C_VEL
LIN {X 0,Y 401.443,Z 759.303,A -85,B 0,C 180,E1 15442.939,E2 15442.939} C_VEL
LIN {X 0,Y 397.887,Z 781.661,A -85,B 0,C 180,E1 15442.102,E2 15442.102} C_VEL
LIN {X 0,Y 393.849,Z 802.386,A -85,B 0,C 180,E1 15441.092,E2 15441.092} C_VEL
LIN {X 0,Y 388.971,Z 824.168,A -85,B 0,C 180,E1 15439.773,E2 15439.773} C_VEL
LIN {X 0,Y 384.074,Z 843.365,A -85,B 0,C 180,E1 15438.348,E2 15438.348} C_VEL
LIN {X 0,Y 378.094,Z 864.781,A -85,B 0,C 180,E1 15436.439,E2 15436.439} C_VEL
LIN {X 0,Y 372.461,Z 883.474,A -85,B 0,C 180,E1 15434.434,E2 15434.434} C_VEL
LIN {X 0,Y 366.531,Z 902.103,A -85,B 0,C 180,E1 15432.059,E2 15432.059} C_VEL
LIN {X 0,Y 360.969,Z 919.093,A -85,B 0,C 180,E1 15429.514,E2 15429.514} C_VEL
LIN {X 0,Y 355.781,Z 934.553,A -85,B 0,C 180,E1 15426.774,E2 15426.774} C_VEL
LIN {X 0,Y 350.92,Z 949.489,A -85,B 0,C 180,E1 15423.698,E2 15423.698} C_VEL
LIN {X 0,Y 346.549,Z 963.181,A -85,B 0,C 180,E1 15420.33,E2 15420.33} C_VEL
LIN {X 0,Y 342.869,Z 975.727,A -85,B 0,C 180,E1 15416.69,E2 15416.69} C_VEL
LIN {X 0,Y 340.227,Z 985.805,A -85,B 0,C 180,E1 15413.196,E2 15413.196} C_VEL
LIN {X 0,Y 338.201,Z 995.006,A -85,B 0,C 180,E1 15409.341,E2 15409.341} C_VEL
LIN {X 0,Y 337.02,Z 1001.803,A -85,B 0,C 180,E1 15405.844,E2 15405.844} C_VEL
LIN {X 0,Y 336.267,Z 1007.85,A -85,B 0,C 180,E1 15401.844,E2 15401.844} C_VEL
LIN {X 0,Y 336.028,Z 1011.671,A -85,B 0,C 180,E1 15398.389,E2 15398.389} C_VEL
LIN {X 0,Y 335.938,Z 1014.381,A -85,B 0,C 180,E1 15394.614,E2 15394.614} C_VEL
LIN {X 0,Y 335.947,Z 1015.426,A -85,B 0,C 180,E1 15391.369,E2 15391.369} C_VEL
LIN {X 0,Y 335.949,Z 1015.377,A -85,B 0,C 180,E1 15388.129,E2 15388.129} C_VEL
LIN {X 0,Y 335.943,Z 1013.872,A -85,B 0,C 180,E1 15384.369,E2 15384.369} C_VEL
LIN {X 0,Y 336.05,Z 1011.13,A -85,B 0,C 180,E1 15380.933,E2 15380.933} C_VEL
LIN {X 0,Y 336.424,Z 1006.663,A -85,B 0,C 180,E1 15377.112,E2 15377.112} C_VEL
LIN {X 0,Y 337.22,Z 1000.786,A -85,B 0,C 180,E1 15373.469,E2 15373.469} C_VEL
LIN {X 0,Y 338.687,Z 993.027,A -85,B 0,C 180,E1 15369.62,E2 15369.62} C_VEL
LIN {X 0,Y 340.72,Z 984.266,A -85,B 0,C 180,E1 15366.118,E2 15366.118} C_VEL
LIN {X 0,Y 343.691,Z 973.353,A -85,B 0,C 180,E1 15362.455,E2 15362.455} C_VEL
LIN {X 0,Y 347.274,Z 961.341,A -85,B 0,C 180,E1 15359.09,E2 15359.09} C_VEL
LIN {X 0,Y 351.766,Z 947.279,A -85,B 0,C 180,E1 15355.758,E2 15355.758} C_VEL
LIN {X 0,Y 356.395,Z 933.172,A -85,B 0,C 180,E1 15352.91,E2 15352.91} C_VEL
LIN {X 0,Y 361.882,Z 916.459,A -85,B 0,C 180,E1 15350.056,E2 15350.056} C_VEL
LIN {X 0,Y 367.423,Z 899.356,A -85,B 0,C 180,E1 15347.564,E2 15347.564} C_VEL
LIN {X 0,Y 373.094,Z 880.797,A -85,B 0,C 180,E1 15345.302,E2 15345.302} C_VEL
LIN {X 0,Y 378.867,Z 860.931,A -85,B 0,C 180,E1 15343.258,E2 15343.258} C_VEL
LIN {X 0,Y 383.885,Z 841.947,A -85,B 0,C 180,E1 15341.634,E2 15341.634} C_VEL
LIN {X 0,Y 389.205,Z 819.636,A -85,B 0,C 180,E1 15340.053,E2 15340.053} C_VEL
LIN {X 0,Y 393.257,Z 800.154,A -85,B 0,C 180,E1 15338.931,E2 15338.931} C_VEL
LIN {X 0,Y 397.404,Z 776.507,A -85,B 0,C 180,E1 15337.85,E2 15337.85} C_VEL
LIN {X 0,Y 400.36,Z 755.804,A -85,B 0,C 180,E1 15337.13,E2 15337.13} C_VEL
LIN {X 0,Y 402.77,Z 731.553,A -85,B 0,C 180,E1 15336.511,E2 15336.511} C_VEL
LIN {X 0,Y 414.413,Z 523.569,A -85,B 0,C 180,E1 15332.423,E2 15332.423} C_VEL
LIN {X 0,Y 416.28,Z 489.875,A -85,B 0,C 180,E1 15331.736,E2 15331.736} C_VEL
LIN {X 0,Y 406.651,Z 474.521,A -85,B 0,C 180,E1 15329.132,E2 15329.132} C_VEL
LIN {X 0,Y 397.261,Z 460.435,A -85,B 0,C 180,E1 15326.333,E2 15326.333} C_VEL
LIN {X 0,Y 390.521,Z 451.026,A -85,B 0,C 180,E1 15324.142,E2 15324.142} C_VEL
LIN {X 0,Y 384.732,Z 443.194,A -85,B 0,C 180,E1 15322.097,E2 15322.097} C_VEL
LIN {X 0,Y 381.316,Z 438.816,A -85,B 0,C 180,E1 15320.811,E2 15320.811} C_VEL
LIN {X 0,Y 376.873,Z 433.387,A -85,B 0,C 180,E1 15319.045,E2 15319.045} C_VEL
LIN {X 0,Y 373.167,Z 428.864,A -85,B 0,C 180,E1 15317.462,E2 15317.462} C_VEL
LIN {X 0,Y 368.382,Z 423.384,A -85,B 0,C 180,E1 15315.264,E2 15315.264} C_VEL
LIN {X 0,Y 367.202,Z 421.774,A -85,B 0,C 180,E1 15314.668,E2 15314.668} C_VEL
LIN {X 0,Y 363.791,Z 418.495,A -85,B 0,C 180,E1 15312.943,E2 15312.943} C_VEL
LIN {X 0,Y 362.089,Z 415.705,A -85,B 0,C 180,E1 15311.952,E2 15311.952} C_VEL
LIN {X 0,Y 358.474,Z 412.69,A -85,B 0,C 180,E1 15309.876,E2 15309.876} C_VEL
LIN {X 0,Y 356.301,Z 409.191,A -85,B 0,C 180,E1 15308.39,E2 15308.39} C_VEL
LIN {X 0,Y 352.725,Z 406.563,A -85,B 0,C 180,E1 15305.938,E2 15305.938} C_VEL
LIN {X 0,Y 350.639,Z 402.876,A -85,B 0,C 180,E1 15304.087,E2 15304.087} C_VEL
LIN {X 0,Y 346.249,Z 399.734,A -85,B 0,C 180,E1 15299.999,E2 15299.999} C_VEL
LIN {X 0,Y 344.288,Z 396.212,A -85,B 0,C 180,E1 15297.304,E2 15297.304} C_VEL
LIN {X 0,Y 340.755,Z 394.069,A -85,B 0,C 180,E1 15290.712,E2 15290.712} C_VEL
LIN {X 0,Y 339.946,Z 393.307,A -85,B 0,C 180,E1 15285.347,E2 15285.347} C_VEL
LIN {X 0,Y 340.893,Z 394.196,A -85,B 0,C 180,E1 15280.108,E2 15280.108} C_VEL
LIN {X 0,Y 344.213,Z 396.143,A -85,B 0,C 180,E1 15273.983,E2 15273.983} C_VEL
LIN {X 0,Y 345.37,Z 398.186,A -85,B 0,C 180,E1 15272.345,E2 15272.345} C_VEL
LIN {X 0,Y 347.82,Z 401.24,A -85,B 0,C 180,E1 15269.606,E2 15269.606} C_VEL
LIN {X 0,Y 350.905,Z 403.15,A -85,B 0,C 180,E1 15266.93,E2 15266.93} C_VEL
LIN {X 0,Y 352.792,Z 406.578,A -85,B 0,C 180,E1 15265.273,E2 15265.273} C_VEL
LIN {X 0,Y 356.026,Z 409.051,A -85,B 0,C 180,E1 15263.058,E2 15263.058} C_VEL
LIN {X 0,Y 356.797,Z 409.754,A -85,B 0,C 180,E1 15262.547,E2 15262.547} C_VEL
LIN {X 0,Y 358.954,Z 413.249,A -85,B 0,C 180,E1 15261.087,E2 15261.087} C_VEL
LIN {X 0,Y 362.384,Z 416.111,A -85,B 0,C 180,E1 15259.162,E2 15259.162} C_VEL
LIN {X 0,Y 365.102,Z 420.019,A -85,B 0,C 180,E1 15257.647,E2 15257.647} C_VEL
LIN {X 0,Y 367.887,Z 422.519,A -85,B 0,C 180,E1 15256.289,E2 15256.289} C_VEL
LIN {X 0,Y 371.241,Z 426.872,A -85,B 0,C 180,E1 15254.68,E2 15254.68} C_VEL
LIN {X 0,Y 373.092,Z 428.724,A -85,B 0,C 180,E1 15253.87,E2 15253.87} C_VEL
LIN {X 0,Y 376.684,Z 433.185,A -85,B 0,C 180,E1 15252.332,E2 15252.332} C_VEL
LIN {X 0,Y 378.564,Z 435.511,A -85,B 0,C 180,E1 15251.566,E2 15251.566} C_VEL
LIN {X 0,Y 383.093,Z 441.01,A -85,B 0,C 180,E1 15249.826,E2 15249.826} C_VEL
LIN {X 0,Y 388.331,Z 447.546,A -85,B 0,C 180,E1 15247.958,E2 15247.958} C_VEL
LIN {X 0,Y 394.963,Z 455.967,A -85,B 0,C 180,E1 15245.771,E2 15245.771} C_VEL
LIN {X 0,Y 405.449,Z 470.19,A -85,B 0,C 180,E1 15242.643,E2 15242.643} C_VEL
LIN {X 0,Y 415.611,Z 484.965,A -85,B 0,C 180,E1 15239.918,E2 15239.918} C_VEL
LIN {X 0,Y 416.059,Z 486.065,A -85,B 0,C 180,E1 15239.79,E2 15239.79} C_VEL
LIN {X 0,Y 404.345,Z 694.034,A -85,B 0,C 180,E1 15235.722,E2 15235.722} C_VEL
LIN {X 0,Y 402.217,Z 723.832,A -85,B 0,C 180,E1 15235.071,E2 15235.071} C_VEL
LIN {X 0,Y 399.619,Z 746.444,A -85,B 0,C 180,E1 15234.377,E2 15234.377} C_VEL
LIN {X 0,Y 396.194,Z 768.514,A -85,B 0,C 180,E1 15233.454,E2 15233.454} C_VEL
LIN {X 0,Y 392.208,Z 790.079,A -85,B 0,C 180,E1 15232.318,E2 15232.318} C_VEL
LIN {X 0,Y 387.744,Z 810.153,A -85,B 0,C 180,E1 15230.998,E2 15230.998} C_VEL
LIN {X 0,Y 382.652,Z 830.699,A -85,B 0,C 180,E1 15229.375,E2 15229.375} C_VEL
LIN {X 0,Y 377.38,Z 849.561,A -85,B 0,C 180,E1 15227.575,E2 15227.575} C_VEL
LIN {X 0,Y 371.502,Z 869.003,A -85,B 0,C 180,E1 15225.368,E2 15225.368} C_VEL
LIN {X 0,Y 366.095,Z 885.83,A -85,B 0,C 180,E1 15223.097,E2 15223.097} C_VEL
LIN {X 0,Y 360.402,Z 902.807,A -85,B 0,C 180,E1 15220.384,E2 15220.384} C_VEL
LIN {X 0,Y 359.956,Z 904.101,A -85,B 0,C 180,E1 15220.156,E2 15220.156} C_VEL
LIN {X 0,Y 357.366,Z 909.368,A -85,B 0,C 180,E1 15219.323,E2 15219.323} C_VEL
LIN {X 0,Y 347.845,Z 922.184,A -85,B 0,C 180,E1 15217.341,E2 15217.341} C_VEL
LIN {X 0,Y 345.359,Z 926.835,A -85,B 0,C 180,E1 15216.41,E2 15216.41} C_VEL
LIN {X 0,Y 340.798,Z 939.606,A -85,B 0,C 180,E1 15213.19,E2 15213.19} C_VEL
LIN {X 0,Y 336.783,Z 951.523,A -85,B 0,C 180,E1 15209.655,E2 15209.655} C_VEL
LIN {X 0,Y 333.609,Z 961.513,A -85,B 0,C 180,E1 15206.042,E2 15206.042} C_VEL
LIN {X 0,Y 331.176,Z 970.397,A -85,B 0,C 180,E1 15202.187,E2 15202.187} C_VEL
LIN {X 0,Y 329.604,Z 977.205,A -85,B 0,C 180,E1 15198.475,E2 15198.475} C_VEL
LIN {X 0,Y 328.607,Z 982.989,A -85,B 0,C 180,E1 15194.464,E2 15194.464} C_VEL
LIN {X 0,Y 328.16,Z 986.637,A -85,B 0,C 180,E1 15190.968,E2 15190.968} C_VEL
LIN {X 0,Y 328.002,Z 989.211,A -85,B 0,C 180,E1 15187.408,E2 15187.408} C_VEL
LIN {X 0,Y 327.94,Z 990.491,A -85,B 0,C 180,E1 15183.688,E2 15183.688} C_VEL
LIN {X 0,Y 327.945,Z 990.541,A -85,B 0,C 180,E1 15180.397,E2 15180.397} C_VEL
LIN {X 0,Y 327.995,Z 989.441,A -85,B 0,C 180,E1 15176.717,E2 15176.717} C_VEL
LIN {X 0,Y 328.167,Z 986.824,A -85,B 0,C 180,E1 15172.966,E2 15172.966} C_VEL
LIN {X 0,Y 328.676,Z 983.001,A -85,B 0,C 180,E1 15169.243,E2 15169.243} C_VEL
LIN {X 0,Y 329.69,Z 977.294,A -85,B 0,C 180,E1 15165.279,E2 15165.279} C_VEL
LIN {X 0,Y 331.334,Z 970.511,A -85,B 0,C 180,E1 15161.544,E2 15161.544} C_VEL
LIN {X 0,Y 333.8,Z 961.79,A -85,B 0,C 180,E1 15157.736,E2 15157.736} C_VEL
LIN {X 0,Y 337.077,Z 951.837,A -85,B 0,C 180,E1 15154.1,E2 15154.1} C_VEL
LIN {X 0,Y 341.055,Z 940.435,A -85,B 0,C 180,E1 15150.672,E2 15150.672} C_VEL
LIN {X 0,Y 346.023,Z 927.002,A -85,B 0,C 180,E1 15147.249,E2 15147.249} C_VEL
LIN {X 0,Y 351.137,Z 913.303,A -85,B 0,C 180,E1 15144.322,E2 15144.322} C_VEL
LIN {X 0,Y 357.356,Z 896.511,A -85,B 0,C 180,E1 15141.289,E2 15141.289} C_VEL
LIN {X 0,Y 363.321,Z 880.033,A -85,B 0,C 180,E1 15138.784,E2 15138.784} C_VEL
LIN {X 0,Y 369.346,Z 862.251,A -85,B 0,C 180,E1 15136.514,E2 15136.514} C_VEL
LIN {X 0,Y 375.289,Z 843.697,A -85,B 0,C 180,E1 15134.504,E2 15134.504} C_VEL
LIN {X 0,Y 380.95,Z 823.972,A -85,B 0,C 180,E1 15132.737,E2 15132.737} C_VEL
LIN {X 0,Y 386.472,Z 802.608,A -85,B 0,C 180,E1 15131.151,E2 15131.151} C_VEL
LIN {X 0,Y 391.061,Z 782.032,A -85,B 0,C 180,E1 15129.911,E2 15129.911} C_VEL
LIN {X 0,Y 395.374,Z 758.793,A -85,B 0,C 180,E1 15128.801,E2 15128.801} C_VEL
LIN {X 0,Y 398.621,Z 736.857,A -85,B 0,C 180,E1 15127.998,E2 15127.998} C_VEL
LIN {X 0,Y 401.037,Z 713.756,A -85,B 0,C 180,E1 15127.391,E2 15127.391} C_VEL
LIN {X 0,Y 415.538,Z 503.322,A -85,B 0,C 180,E1 15123.115,E2 15123.115} C_VEL
LIN {X 0,Y 416.339,Z 491.536,A -85,B 0,C 180,E1 15122.857,E2 15122.857} C_VEL
LIN {X 0,Y 409.97,Z 480.99,A -85,B 0,C 180,E1 15120.477,E2 15120.477} C_VEL
LIN {X 0,Y 404.451,Z 472.372,A -85,B 0,C 180,E1 15118.017,E2 15118.017} C_VEL
LIN {X 0,Y 401.086,Z 467.407,A -85,B 0,C 180,E1 15116.213,E2 15116.213} C_VEL
LIN {X 0,Y 398.273,Z 463.107,A -85,B 0,C 180,E1 15114.382,E2 15114.382} C_VEL
LIN {X 0,Y 395.557,Z 459.095,A -85,B 0,C 180,E1 15112.082,E2 15112.082} C_VEL
LIN {X 0,Y 395.085,Z 458.157,A -85,B 0,C 180,E1 15111.56,E2 15111.56} C_VEL
LIN {X 0,Y 392.659,Z 455.279,A -85,B 0,C 180,E1 15106.902,E2 15106.902} C_VEL
LIN {X 0,Y 392.766,Z 455.557,A -85,B 0,C 180,E1 15104.8,E2 15104.8} C_VEL
LIN {X 0,Y 395.349,Z 458.601,A -85,B 0,C 180,E1 15100.576,E2 15100.576} C_VEL
LIN {X 0,Y 397.788,Z 462.659,A -85,B 0,C 180,E1 15098.394,E2 15098.394} C_VEL
LIN {X 0,Y 398.908,Z 464.106,A -85,B 0,C 180,E1 15097.606,E2 15097.606} C_VEL
LIN {X 0,Y 402.448,Z 469.568,A -85,B 0,C 180,E1 15095.448,E2 15095.448} C_VEL
LIN {X 0,Y 406.935,Z 477.387,A -85,B 0,C 180,E1 15093.201,E2 15093.201} C_VEL
LIN {X 0,Y 412.134,Z 486.794,A -85,B 0,C 180,E1 15091.014,E2 15091.014} C_VEL
LIN {X 0,Y 416.318,Z 495.024,A -85,B 0,C 180,E1 15089.458,E2 15089.458} C_VEL
LIN {X 0,Y 403.263,Z 684.856,A -85,B 0,C 180,E1 15085.603,E2 15085.603} C_VEL
LIN {X 0,Y 399.742,Z 736.085,A -85,B 0,C 180,E1 15084.536,E2 15084.536} C_VEL
LIN {X 0,Y 396.835,Z 758.918,A -85,B 0,C 180,E1 15083.891,E2 15083.891} C_VEL
LIN {X 0,Y 393.013,Z 782.004,A -85,B 0,C 180,E1 15083.024,E2 15083.024} C_VEL
LIN {X 0,Y 389.108,Z 801.303,A -85,B 0,C 180,E1 15082.085,E2 15082.085} C_VEL
LIN {X 0,Y 384.184,Z 822.634,A -85,B 0,C 180,E1 15080.804,E2 15080.804} C_VEL
LIN {X 0,Y 378.872,Z 842.7,A -85,B 0,C 180,E1 15079.32,E2 15079.32} C_VEL
LIN {X 0,Y 372.926,Z 863.205,A -85,B 0,C 180,E1 15077.497,E2 15077.497} C_VEL
LIN {X 0,Y 367.126,Z 881.628,A -85,B 0,C 180,E1 15075.529,E2 15075.529} C_VEL
LIN {X 0,Y 360.561,Z 901.34,A -85,B 0,C 180,E1 15073.018,E2 15073.018} C_VEL
LIN {X 0,Y 354.717,Z 918.383,A -85,B 0,C 180,E1 15070.443,E2 15070.443} C_VEL
LIN {X 0,Y 349.099,Z 934.248,A -85,B 0,C 180,E1 15067.598,E2 15067.598} C_VEL
LIN {X 0,Y 344.046,Z 948.953,A -85,B 0,C 180,E1 15064.525,E2 15064.525} C_VEL
LIN {X 0,Y 339.528,Z 962.202,A -85,B 0,C 180,E1 15061.222,E2 15061.222} C_VEL
LIN {X 0,Y 335.743,Z 974.336,A -85,B 0,C 180,E1 15057.687,E2 15057.687} C_VEL
LIN {X 0,Y 332.758,Z 984.802,A -85,B 0,C 180,E1 15054.015,E2 15054.015} C_VEL
LIN {X 0,Y 330.476,Z 994.315,A -85,B 0,C 180,E1 15049.996,E2 15049.996} C_VEL
LIN {X 0,Y 329.133,Z 1001.419,A -85,B 0,C 180,E1 15046.27,E2 15046.27} C_VEL
LIN {X 0,Y 328.306,Z 1007.515,A -85,B 0,C 180,E1 15042.151,E2 15042.151} C_VEL
LIN {X 0,Y 328.036,Z 1011.362,A -85,B 0,C 180,E1 15038.594,E2 15038.594} C_VEL
LIN {X 0,Y 327.942,Z 1014.077,A -85,B 0,C 180,E1 15034.727,E2 15034.727} C_VEL
LIN {X 0,Y 327.952,Z 1015.125,A -85,B 0,C 180,E1 15031.403,E2 15031.403} C_VEL
LIN {X 0,Y 327.953,Z 1015.101,A -85,B 0,C 180,E1 15028.258,E2 15028.258} C_VEL
LIN {X 0,Y 327.945,Z 1013.687,A -85,B 0,C 180,E1 15024.407,E2 15024.407} C_VEL
LIN {X 0,Y 328.053,Z 1010.989,A -85,B 0,C 180,E1 15020.887,E2 15020.887} C_VEL
LIN {X 0,Y 328.441,Z 1006.628,A -85,B 0,C 180,E1 15016.987,E2 15016.987} C_VEL
LIN {X 0,Y 329.281,Z 1000.775,A -85,B 0,C 180,E1 15013.24,E2 15013.24} C_VEL
LIN {X 0,Y 330.829,Z 993.108,A -85,B 0,C 180,E1 15009.298,E2 15009.298} C_VEL
LIN {X 0,Y 333.099,Z 983.914,A -85,B 0,C 180,E1 15005.536,E2 15005.536} C_VEL
